Fanuc TP program (LS listing): ultrahose3.ls

/PROG  ultrahose3
/ATTR
COMMENT	= "19-03-19 19:07:18";
PROG_SIZE	= 0;
DEFAULT_GROUP	= 1, *, *, *, *;
/APPL
    ARC Welding Equipment: 1, *, *, *, *;
/MN
   1:  CALL HOME_ALL;
   1:  UFRAME_NUM = 1;
   1:  UTOOL_NUM = 3;
   1:  COL GUARD ADJUST 150;
   1:  PR[91] = PR[90];
   1:  PR[91,1] = PR[90,1] + -62.704;
   1:  PR[91,2] = PR[90,2] + 18.714;
   1:  PR[91,3] = PR[90,3] + 69.095;
   1:L PR[91] R[100]mm/sec CNT100;
   1:  PR[91,1] = PR[90,1] + -67.808;
   1:  PR[91,2] = PR[90,2] + 15.587;
   1:  PR[91,3] = PR[90,3] + 67.803;
   1:L PR[91] R[100]mm/sec CNT100;
   1:  PR[91,1] = PR[90,1] + -70.681;
   1:  PR[91,2] = PR[90,2] + 12.957;
   1:  PR[91,3] = PR[90,3] + 67.824;
   1:L PR[91] R[100]mm/sec CNT100;
   1:  PR[91,1] = PR[90,1] + -71.666;
   1:  PR[91,2] = PR[90,2] + 11.982;
   1:  PR[91,3] = PR[90,3] + 67.838;
   1:L PR[91] R[100]mm/sec CNT100;
   1:  PR[91,1] = PR[90,1] + -74.314;
   1:  PR[91,2] = PR[90,2] + 7.950;
   1:  PR[91,3] = PR[90,3] + 67.843;
   1:L PR[91] R[100]mm/sec CNT100;
   1:  PR[91,1] = PR[90,1] + -75.904;
   1:  PR[91,2] = PR[90,2] + 3.669;
   1:  PR[91,3] = PR[90,3] + 67.861;
   1:L PR[91] R[100]mm/sec CNT100;
   1:  PR[91,1] = PR[90,1] + -76.068;
   1:  PR[91,2] = PR[90,2] + 2.308;
   1:  PR[91,3] = PR[90,3] + 67.877;
   1:L PR[91] R[100]mm/sec CNT100;
   1:  PR[91,1] = PR[90,1] + -76.476;
   1:  PR[91,2] = PR[90,2] + 0.036;
   1:  PR[91,3] = PR[90,3] + 67.882;
   1:L PR[91] R[100]mm/sec CNT100;
   1:  PR[91,1] = PR[90,1] + -76.570;
   1:  PR[91,2] = PR[90,2] + -0.724;
   1:  PR[91,3] = PR[90,3] + 67.890;
   1:L PR[91] R[100]mm/sec CNT100;
   1:  PR[91,1] = PR[90,1] + -76.127;
   1:  PR[91,2] = PR[90,2] + -4.152;
   1:  PR[91,3] = PR[90,3] + 67.893;
   1:L PR[91] R[100]mm/sec CNT100;
   1:  PR[91,1] = PR[90,1] + -75.971;
   1:  PR[91,2] = PR[90,2] + -4.906;
   1:  PR[91,3] = PR[90,3] + 67.905;
   1:L PR[91] R[100]mm/sec CNT100;
   1:  PR[91,1] = PR[90,1] + -75.920;
   1:  PR[91,2] = PR[90,2] + -5.300;
   1:  PR[91,3] = PR[90,3] + 67.908;
   1:L PR[91] R[100]mm/sec CNT100;
   1:  PR[91,1] = PR[90,1] + -74.122;
   1:  PR[91,2] = PR[90,2] + -9.726;
   1:  PR[91,3] = PR[90,3] + 67.910;
   1:L PR[91] R[100]mm/sec CNT100;
   1:  PR[91,1] = PR[90,1] + -71.147;
   1:  PR[91,2] = PR[90,2] + -13.861;
   1:  PR[91,3] = PR[90,3] + 67.927;
   1:L PR[91] R[100]mm/sec CNT100;
   1:  PR[91,1] = PR[90,1] + -69.141;
   1:  PR[91,2] = PR[90,2] + -15.680;
   1:  PR[91,3] = PR[90,3] + 67.945;
   1:L PR[91] R[100]mm/sec CNT100;
   1:  PR[91,1] = PR[90,1] + -67.080;
   1:  PR[91,2] = PR[90,2] + -17.518;
   1:  PR[91,3] = PR[90,3] + 67.955;
   1:L PR[91] R[100]mm/sec CNT100;
   1:  PR[91,1] = PR[90,1] + -62.025;
   1:  PR[91,2] = PR[90,2] + -20.541;
   1:  PR[91,3] = PR[90,3] + 67.965;
   1:L PR[91] R[100]mm/sec CNT100;
   1:  PR[91,1] = PR[90,1] + -60.674;
   1:  PR[91,2] = PR[90,2] + -21.047;
   1:  PR[91,3] = PR[90,3] + 67.986;
   1:L PR[91] R[100]mm/sec CNT100;
   1:  PR[91,1] = PR[90,1] + -56.313;
   1:  PR[91,2] = PR[90,2] + -22.600;
   1:  PR[91,3] = PR[90,3] + 67.991;
   1:L PR[91] R[100]mm/sec CNT100;
   1:  PR[91,1] = PR[90,1] + -53.537;
   1:  PR[91,2] = PR[90,2] + -23.271;
   1:  PR[91,3] = PR[90,3] + 68.008;
   1:L PR[91] R[100]mm/sec CNT100;
   1:  PR[91,1] = PR[90,1] + -50.510;
   1:  PR[91,2] = PR[90,2] + -23.850;
   1:  PR[91,3] = PR[90,3] + 68.018;
   1:L PR[91] R[100]mm/sec CNT100;
   1:  PR[91,1] = PR[90,1] + -46.666;
   1:  PR[91,2] = PR[90,2] + -24.219;
   1:  PR[91,3] = PR[90,3] + 68.029;
   1:L PR[91] R[100]mm/sec CNT100;
   1:  PR[91,1] = PR[90,1] + -44.723;
   1:  PR[91,2] = PR[90,2] + -24.423;
   1:  PR[91,3] = PR[90,3] + 68.043;
   1:L PR[91] R[100]mm/sec CNT100;
   1:  PR[91,1] = PR[90,1] + -43.071;
   1:  PR[91,2] = PR[90,2] + -24.533;
   1:  PR[91,3] = PR[90,3] + 68.050;
   1:L PR[91] R[100]mm/sec CNT100;
   1:  PR[91,1] = PR[90,1] + -39.194;
   1:  PR[91,2] = PR[90,2] + -24.475;
   1:  PR[91,3] = PR[90,3] + 68.056;
   1:L PR[91] R[100]mm/sec CNT100;
   1:  PR[91,1] = PR[90,1] + -35.228;
   1:  PR[91,2] = PR[90,2] + -24.237;
   1:  PR[91,3] = PR[90,3] + 68.070;
   1:L PR[91] R[100]mm/sec CNT100;
   1:  PR[91,1] = PR[90,1] + -31.937;
   1:  PR[91,2] = PR[90,2] + -24.126;
   1:  PR[91,3] = PR[90,3] + 68.085;
   1:L PR[91] R[100]mm/sec CNT100;
   1:  PR[91,1] = PR[90,1] + -25.421;
   1:  PR[91,2] = PR[90,2] + -23.278;
   1:  PR[91,3] = PR[90,3] + 68.096;
   1:L PR[91] R[100]mm/sec CNT100;
   1:  PR[91,1] = PR[90,1] + -23.909;
   1:  PR[91,2] = PR[90,2] + -23.104;
   1:  PR[91,3] = PR[90,3] + 68.120;
   1:L PR[91] R[100]mm/sec CNT100;
   1:  PR[91,1] = PR[90,1] + -23.194;
   1:  PR[91,2] = PR[90,2] + -22.983;
   1:  PR[91,3] = PR[90,3] + 68.126;
   1:L PR[91] R[100]mm/sec CNT100;
   1:  PR[91,1] = PR[90,1] + -18.760;
   1:  PR[91,2] = PR[90,2] + -22.151;
   1:  PR[91,3] = PR[90,3] + 68.128;
   1:L PR[91] R[100]mm/sec CNT100;
   1:  PR[91,1] = PR[90,1] + -17.454;
   1:  PR[91,2] = PR[90,2] + -22.712;
   1:  PR[91,3] = PR[90,3] + 68.144;
   1:L PR[91] R[100]mm/sec CNT100;
   1:  PR[91,1] = PR[90,1] + -16.961;
   1:  PR[91,2] = PR[90,2] + -22.855;
   1:  PR[91,3] = PR[90,3] + 68.150;
   1:L PR[91] R[100]mm/sec CNT100;
   1:  PR[91,1] = PR[90,1] + -14.286;
   1:  PR[91,2] = PR[90,2] + -23.568;
   1:  PR[91,3] = PR[90,3] + 68.151;
   1:L PR[91] R[100]mm/sec CNT100;
   1:  PR[91,1] = PR[90,1] + -12.800;
   1:  PR[91,2] = PR[90,2] + -23.980;
   1:  PR[91,3] = PR[90,3] + 68.161;
   1:L PR[91] R[100]mm/sec CNT100;
   1:  PR[91,1] = PR[90,1] + -12.108;
   1:  PR[91,2] = PR[90,2] + -24.142;
   1:  PR[91,3] = PR[90,3] + 68.167;
   1:L PR[91] R[100]mm/sec CNT100;
   1:  PR[91,1] = PR[90,1] + -11.357;
   1:  PR[91,2] = PR[90,2] + -24.214;
   1:  PR[91,3] = PR[90,3] + 68.170;
   1:L PR[91] R[100]mm/sec CNT100;
   1:  PR[91,1] = PR[90,1] + -6.128;
   1:  PR[91,2] = PR[90,2] + -24.637;
   1:  PR[91,3] = PR[90,3] + 68.172;
   1:L PR[91] R[100]mm/sec CNT100;
   1:  PR[91,1] = PR[90,1] + -2.890;
   1:  PR[91,2] = PR[90,2] + -24.354;
   1:  PR[91,3] = PR[90,3] + 68.191;
   1:L PR[91] R[100]mm/sec CNT100;
   1:  PR[91,1] = PR[90,1] + -0.001;
   1:  PR[91,2] = PR[90,2] + -24.062;
   1:  PR[91,3] = PR[90,3] + 68.203;
   1:L PR[91] R[100]mm/sec CNT100;
   1:  PR[91,1] = PR[90,1] + 5.816;
   1:  PR[91,2] = PR[90,2] + -22.408;
   1:  PR[91,3] = PR[90,3] + 68.213;
   1:L PR[91] R[100]mm/sec CNT100;
   1:  PR[91,1] = PR[90,1] + 6.060;
   1:  PR[91,2] = PR[90,2] + -22.335;
   1:  PR[91,3] = PR[90,3] + 68.235;
   1:L PR[91] R[100]mm/sec CNT100;
   1:  PR[91,1] = PR[90,1] + 7.030;
   1:  PR[91,2] = PR[90,2] + -21.873;
   1:  PR[91,3] = PR[90,3] + 68.236;
   1:L PR[91] R[100]mm/sec CNT100;
   1:  PR[91,1] = PR[90,1] + 8.393;
   1:  PR[91,2] = PR[90,2] + -22.591;
   1:  PR[91,3] = PR[90,3] + 68.240;
   1:L PR[91] R[100]mm/sec CNT100;
   1:  PR[91,1] = PR[90,1] + 11.474;
   1:  PR[91,2] = PR[90,2] + -24.006;
   1:  PR[91,3] = PR[90,3] + 68.245;
   1:L PR[91] R[100]mm/sec CNT100;
   1:  PR[91,1] = PR[90,1] + 15.747;
   1:  PR[91,2] = PR[90,2] + -25.170;
   1:  PR[91,3] = PR[90,3] + 68.258;
   1:L PR[91] R[100]mm/sec CNT100;
   1:  PR[91,1] = PR[90,1] + 17.096;
   1:  PR[91,2] = PR[90,2] + -25.461;
   1:  PR[91,3] = PR[90,3] + 68.274;
   1:L PR[91] R[100]mm/sec CNT100;
   1:  PR[91,1] = PR[90,1] + 21.812;
   1:  PR[91,2] = PR[90,2] + -25.653;
   1:  PR[91,3] = PR[90,3] + 68.279;
   1:L PR[91] R[100]mm/sec CNT100;
   1:  PR[91,1] = PR[90,1] + 22.821;
   1:  PR[91,2] = PR[90,2] + -25.620;
   1:  PR[91,3] = PR[90,3] + 68.296;
   1:L PR[91] R[100]mm/sec CNT100;
   1:  PR[91,1] = PR[90,1] + 24.497;
   1:  PR[91,2] = PR[90,2] + -25.365;
   1:  PR[91,3] = PR[90,3] + 68.299;
   1:L PR[91] R[100]mm/sec CNT100;
   1:  PR[91,1] = PR[90,1] + 28.145;
   1:  PR[91,2] = PR[90,2] + -24.676;
   1:  PR[91,3] = PR[90,3] + 68.305;
   1:L PR[91] R[100]mm/sec CNT100;
   1:  PR[91,1] = PR[90,1] + 30.783;
   1:  PR[91,2] = PR[90,2] + -25.399;
   1:  PR[91,3] = PR[90,3] + 68.319;
   1:L PR[91] R[100]mm/sec CNT100;
   1:  PR[91,1] = PR[90,1] + 33.304;
   1:  PR[91,2] = PR[90,2] + -26.004;
   1:  PR[91,3] = PR[90,3] + 68.329;
   1:L PR[91] R[100]mm/sec CNT100;
   1:  PR[91,1] = PR[90,1] + 37.954;
   1:  PR[91,2] = PR[90,2] + -26.647;
   1:  PR[91,3] = PR[90,3] + 68.338;
   1:L PR[91] R[100]mm/sec CNT100;
   1:  PR[91,1] = PR[90,1] + 43.879;
   1:  PR[91,2] = PR[90,2] + -26.624;
   1:  PR[91,3] = PR[90,3] + 68.355;
   1:L PR[91] R[100]mm/sec CNT100;
   1:  PR[91,1] = PR[90,1] + 49.043;
   1:  PR[91,2] = PR[90,2] + -26.009;
   1:  PR[91,3] = PR[90,3] + 68.376;
   1:L PR[91] R[100]mm/sec CNT100;
   1:  PR[91,1] = PR[90,1] + 53.583;
   1:  PR[91,2] = PR[90,2] + -25.090;
   1:  PR[91,3] = PR[90,3] + 68.395;
   1:L PR[91] R[100]mm/sec CNT100;
   1:  PR[91,1] = PR[90,1] + 55.197;
   1:  PR[91,2] = PR[90,2] + -24.588;
   1:  PR[91,3] = PR[90,3] + 68.411;
   1:L PR[91] R[100]mm/sec CNT100;
   1:  PR[91,1] = PR[90,1] + 59.058;
   1:  PR[91,2] = PR[90,2] + -23.334;
   1:  PR[91,3] = PR[90,3] + 68.418;
   1:L PR[91] R[100]mm/sec CNT100;
   1:  PR[91,1] = PR[90,1] + 61.784;
   1:  PR[91,2] = PR[90,2] + -22.074;
   1:  PR[91,3] = PR[90,3] + 68.432;
   1:L PR[91] R[100]mm/sec CNT100;
   1:  PR[91,1] = PR[90,1] + 65.680;
   1:  PR[91,2] = PR[90,2] + -19.965;
   1:  PR[91,3] = PR[90,3] + 68.443;
   1:L PR[91] R[100]mm/sec CNT100;
   1:  PR[91,1] = PR[90,1] + 66.517;
   1:  PR[91,2] = PR[90,2] + -19.431;
   1:  PR[91,3] = PR[90,3] + 68.459;
   1:L PR[91] R[100]mm/sec CNT100;
   1:  PR[91,1] = PR[90,1] + 69.227;
   1:  PR[91,2] = PR[90,2] + -17.197;
   1:  PR[91,3] = PR[90,3] + 68.463;
   1:L PR[91] R[100]mm/sec CNT100;
   1:  PR[91,1] = PR[90,1] + 71.107;
   1:  PR[91,2] = PR[90,2] + -15.516;
   1:  PR[91,3] = PR[90,3] + 68.475;
   1:L PR[91] R[100]mm/sec CNT100;
   1:  PR[91,1] = PR[90,1] + 74.460;
   1:  PR[91,2] = PR[90,2] + -10.836;
   1:  PR[91,3] = PR[90,3] + 68.484;
   1:L PR[91] R[100]mm/sec CNT100;
   1:  PR[91,1] = PR[90,1] + 76.466;
   1:  PR[91,2] = PR[90,2] + -5.850;
   1:  PR[91,3] = PR[90,3] + 68.505;
   1:L PR[91] R[100]mm/sec CNT100;
   1:  PR[91,1] = PR[90,1] + 76.772;
   1:  PR[91,2] = PR[90,2] + -3.531;
   1:  PR[91,3] = PR[90,3] + 68.524;
   1:L PR[91] R[100]mm/sec CNT100;
   1:  PR[91,1] = PR[90,1] + 77.227;
   1:  PR[91,2] = PR[90,2] + -0.700;
   1:  PR[91,3] = PR[90,3] + 68.533;
   1:L PR[91] R[100]mm/sec CNT100;
   1:  PR[91,1] = PR[90,1] + 77.051;
   1:  PR[91,2] = PR[90,2] + 0.647;
   1:  PR[91,3] = PR[90,3] + 68.543;
   1:L PR[91] R[100]mm/sec CNT100;
   1:  PR[91,1] = PR[90,1] + 76.850;
   1:  PR[91,2] = PR[90,2] + 1.446;
   1:  PR[91,3] = PR[90,3] + 68.548;
   1:L PR[91] R[100]mm/sec CNT100;
   1:  PR[91,1] = PR[90,1] + 76.465;
   1:  PR[91,2] = PR[90,2] + 4.394;
   1:  PR[91,3] = PR[90,3] + 68.551;
   1:L PR[91] R[100]mm/sec CNT100;
   1:  PR[91,1] = PR[90,1] + 74.460;
   1:  PR[91,2] = PR[90,2] + 9.378;
   1:  PR[91,3] = PR[90,3] + 68.562;
   1:L PR[91] R[100]mm/sec CNT100;
   1:  PR[91,1] = PR[90,1] + 71.112;
   1:  PR[91,2] = PR[90,2] + 14.052;
   1:  PR[91,3] = PR[90,3] + 68.581;
   1:L PR[91] R[100]mm/sec CNT100;
   1:  PR[91,1] = PR[90,1] + 69.227;
   1:  PR[91,2] = PR[90,2] + 15.739;
   1:  PR[91,3] = PR[90,3] + 68.602;
   1:L PR[91] R[100]mm/sec CNT100;
   1:  PR[91,1] = PR[90,1] + 66.528;
   1:  PR[91,2] = PR[90,2] + 17.965;
   1:  PR[91,3] = PR[90,3] + 68.611;
   1:L PR[91] R[100]mm/sec CNT100;
   1:  PR[91,1] = PR[90,1] + 65.694;
   1:  PR[91,2] = PR[90,2] + 18.497;
   1:  PR[91,3] = PR[90,3] + 68.623;
   1:L PR[91] R[100]mm/sec CNT100;
   1:  PR[91,1] = PR[90,1] + 61.792;
   1:  PR[91,2] = PR[90,2] + 20.612;
   1:  PR[91,3] = PR[90,3] + 68.627;
   1:L PR[91] R[100]mm/sec CNT100;
   1:  PR[91,1] = PR[90,1] + 59.065;
   1:  PR[91,2] = PR[90,2] + 21.873;
   1:  PR[91,3] = PR[90,3] + 68.643;
   1:L PR[91] R[100]mm/sec CNT100;
   1:  PR[91,1] = PR[90,1] + 55.197;
   1:  PR[91,2] = PR[90,2] + 23.129;
   1:  PR[91,3] = PR[90,3] + 68.654;
   1:L PR[91] R[100]mm/sec CNT100;
   1:  PR[91,1] = PR[90,1] + 53.583;
   1:  PR[91,2] = PR[90,2] + 23.631;
   1:  PR[91,3] = PR[90,3] + 68.668;
   1:L PR[91] R[100]mm/sec CNT100;
   1:  PR[91,1] = PR[90,1] + 49.043;
   1:  PR[91,2] = PR[90,2] + 24.550;
   1:  PR[91,3] = PR[90,3] + 68.675;
   1:L PR[91] R[100]mm/sec CNT100;
   1:  PR[91,1] = PR[90,1] + 43.879;
   1:  PR[91,2] = PR[90,2] + 25.165;
   1:  PR[91,3] = PR[90,3] + 68.691;
   1:L PR[91] R[100]mm/sec CNT100;
   1:  PR[91,1] = PR[90,1] + 37.958;
   1:  PR[91,2] = PR[90,2] + 25.189;
   1:  PR[91,3] = PR[90,3] + 68.710;
   1:L PR[91] R[100]mm/sec CNT100;
   1:  PR[91,1] = PR[90,1] + 33.304;
   1:  PR[91,2] = PR[90,2] + 24.545;
   1:  PR[91,3] = PR[90,3] + 68.731;
   1:L PR[91] R[100]mm/sec CNT100;
   1:  PR[91,1] = PR[90,1] + 30.783;
   1:  PR[91,2] = PR[90,2] + 23.940;
   1:  PR[91,3] = PR[90,3] + 68.748;
   1:L PR[91] R[100]mm/sec CNT100;
   1:  PR[91,1] = PR[90,1] + 28.145;
   1:  PR[91,2] = PR[90,2] + 23.217;
   1:  PR[91,3] = PR[90,3] + 68.758;
   1:L PR[91] R[100]mm/sec CNT100;
   1:  PR[91,1] = PR[90,1] + 24.496;
   1:  PR[91,2] = PR[90,2] + 23.906;
   1:  PR[91,3] = PR[90,3] + 68.767;
   1:L PR[91] R[100]mm/sec CNT100;
   1:  PR[91,1] = PR[90,1] + 22.831;
   1:  PR[91,2] = PR[90,2] + 24.160;
   1:  PR[91,3] = PR[90,3] + 68.781;
   1:L PR[91] R[100]mm/sec CNT100;
   1:  PR[91,1] = PR[90,1] + 21.811;
   1:  PR[91,2] = PR[90,2] + 24.194;
   1:  PR[91,3] = PR[90,3] + 68.787;
   1:L PR[91] R[100]mm/sec CNT100;
   1:  PR[91,1] = PR[90,1] + 17.094;
   1:  PR[91,2] = PR[90,2] + 24.002;
   1:  PR[91,3] = PR[90,3] + 68.791;
   1:L PR[91] R[100]mm/sec CNT100;
   1:  PR[91,1] = PR[90,1] + 15.746;
   1:  PR[91,2] = PR[90,2] + 23.711;
   1:  PR[91,3] = PR[90,3] + 68.808;
   1:L PR[91] R[100]mm/sec CNT100;
   1:  PR[91,1] = PR[90,1] + 11.472;
   1:  PR[91,2] = PR[90,2] + 22.546;
   1:  PR[91,3] = PR[90,3] + 68.812;
   1:L PR[91] R[100]mm/sec CNT100;
   1:  PR[91,1] = PR[90,1] + 8.412;
   1:  PR[91,2] = PR[90,2] + 21.143;
   1:  PR[91,3] = PR[90,3] + 68.828;
   1:L PR[91] R[100]mm/sec CNT100;
   1:  PR[91,1] = PR[90,1] + 7.033;
   1:  PR[91,2] = PR[90,2] + 20.424;
   1:  PR[91,3] = PR[90,3] + 68.841;
   1:L PR[91] R[100]mm/sec CNT100;
   1:  PR[91,1] = PR[90,1] + 6.058;
   1:  PR[91,2] = PR[90,2] + 20.878;
   1:  PR[91,3] = PR[90,3] + 68.846;
   1:L PR[91] R[100]mm/sec CNT100;
   1:  PR[91,1] = PR[90,1] + 5.788;
   1:  PR[91,2] = PR[90,2] + 20.959;
   1:  PR[91,3] = PR[90,3] + 68.850;
   1:L PR[91] R[100]mm/sec CNT100;
   1:  PR[91,1] = PR[90,1] + 0.034;
   1:  PR[91,2] = PR[90,2] + 22.597;
   1:  PR[91,3] = PR[90,3] + 68.851;
   1:L PR[91] R[100]mm/sec CNT100;
   1:  PR[91,1] = PR[90,1] + -2.850;
   1:  PR[91,2] = PR[90,2] + 22.890;
   1:  PR[91,3] = PR[90,3] + 68.873;
   1:L PR[91] R[100]mm/sec CNT100;
   1:  PR[91,1] = PR[90,1] + -6.112;
   1:  PR[91,2] = PR[90,2] + 23.178;
   1:  PR[91,3] = PR[90,3] + 68.883;
   1:L PR[91] R[100]mm/sec CNT100;
   1:  PR[91,1] = PR[90,1] + -11.344;
   1:  PR[91,2] = PR[90,2] + 22.757;
   1:  PR[91,3] = PR[90,3] + 68.895;
   1:L PR[91] R[100]mm/sec CNT100;
   1:  PR[91,1] = PR[90,1] + -12.102;
   1:  PR[91,2] = PR[90,2] + 22.684;
   1:  PR[91,3] = PR[90,3] + 68.914;
   1:L PR[91] R[100]mm/sec CNT100;
   1:  PR[91,1] = PR[90,1] + -12.809;
   1:  PR[91,2] = PR[90,2] + 22.518;
   1:  PR[91,3] = PR[90,3] + 68.916;
   1:L PR[91] R[100]mm/sec CNT100;
   1:  PR[91,1] = PR[90,1] + -14.290;
   1:  PR[91,2] = PR[90,2] + 22.107;
   1:  PR[91,3] = PR[90,3] + 68.919;
   1:L PR[91] R[100]mm/sec CNT100;
   1:  PR[91,1] = PR[90,1] + -16.962;
   1:  PR[91,2] = PR[90,2] + 21.395;
   1:  PR[91,3] = PR[90,3] + 68.925;
   1:L PR[91] R[100]mm/sec CNT100;
   1:  PR[91,1] = PR[90,1] + -17.452;
   1:  PR[91,2] = PR[90,2] + 21.253;
   1:  PR[91,3] = PR[90,3] + 68.935;
   1:L PR[91] R[100]mm/sec CNT100;
   1:  PR[91,1] = PR[90,1] + -18.760;
   1:  PR[91,2] = PR[90,2] + 20.692;
   1:  PR[91,3] = PR[90,3] + 68.936;
   1:L PR[91] R[100]mm/sec CNT100;
   1:  PR[91,1] = PR[90,1] + -23.191;
   1:  PR[91,2] = PR[90,2] + 21.523;
   1:  PR[91,3] = PR[90,3] + 68.942;
   1:L PR[91] R[100]mm/sec CNT100;
   1:  PR[91,1] = PR[90,1] + -23.903;
   1:  PR[91,2] = PR[90,2] + 21.644;
   1:  PR[91,3] = PR[90,3] + 68.958;
   1:L PR[91] R[100]mm/sec CNT100;
   1:  PR[91,1] = PR[90,1] + -25.418;
   1:  PR[91,2] = PR[90,2] + 21.819;
   1:  PR[91,3] = PR[90,3] + 68.960;
   1:L PR[91] R[100]mm/sec CNT100;
   1:  PR[91,1] = PR[90,1] + -32.341;
   1:  PR[91,2] = PR[90,2] + 22.697;
   1:  PR[91,3] = PR[90,3] + 68.966;
   1:L PR[91] R[100]mm/sec CNT100;
   1:  PR[91,1] = PR[90,1] + -34.160;
   1:  PR[91,2] = PR[90,2] + 22.753;
   1:  PR[91,3] = PR[90,3] + 68.991;
   1:L PR[91] R[100]mm/sec CNT100;
   1:  PR[91,1] = PR[90,1] + -39.829;
   1:  PR[91,2] = PR[90,2] + 23.076;
   1:  PR[91,3] = PR[90,3] + 68.998;
   1:L PR[91] R[100]mm/sec CNT100;
   1:  PR[91,1] = PR[90,1] + -44.279;
   1:  PR[91,2] = PR[90,2] + 22.883;
   1:  PR[91,3] = PR[90,3] + 69.018;
   1:L PR[91] R[100]mm/sec CNT100;
   1:  PR[91,1] = PR[90,1] + -46.346;
   1:  PR[91,2] = PR[90,2] + 22.848;
   1:  PR[91,3] = PR[90,3] + 69.034;
   1:L PR[91] R[100]mm/sec CNT100;
   1:  PR[91,1] = PR[90,1] + -47.984;
   1:  PR[91,2] = PR[90,2] + 22.746;
   1:  PR[91,3] = PR[90,3] + 69.042;
   1:L PR[91] R[100]mm/sec CNT100;
   1:  PR[91,1] = PR[90,1] + -51.432;
   1:  PR[91,2] = PR[90,2] + 22.175;
   1:  PR[91,3] = PR[90,3] + 69.047;
   1:L PR[91] R[100]mm/sec CNT100;
   1:  PR[91,1] = PR[90,1] + -56.575;
   1:  PR[91,2] = PR[90,2] + 21.118;
   1:  PR[91,3] = PR[90,3] + 69.060;
   1:L PR[91] R[100]mm/sec CNT100;
   1:  PR[91,1] = PR[90,1] + -56.591;
   1:  PR[91,2] = PR[90,2] + 21.114;
   1:  PR[91,3] = PR[90,3] + 69.079;
   1:L PR[91] R[100]mm/sec CNT100;
   1:  PR[91,1] = PR[90,1] + -60.733;
   1:  PR[91,2] = PR[90,2] + 19.500;
   1:L PR[91] R[100]mm/sec CNT100;
   1:  PR[91] = PR[90];
   1:  PR[91,1] = PR[90,1] + -66.757;
   1:  PR[91,2] = PR[90,2] + 15.737;
   1:  PR[91,3] = PR[90,3] + 70.395;
   1:L PR[91] R[100]mm/sec CNT100;
   1:  PR[91,1] = PR[90,1] + -70.803;
   1:  PR[91,2] = PR[90,2] + 12.036;
   1:  PR[91,3] = PR[90,3] + 69.117;
   1:L PR[91] R[100]mm/sec CNT100;
   1:  PR[91,1] = PR[90,1] + -72.056;
   1:  PR[91,2] = PR[90,2] + 10.273;
   1:  PR[91,3] = PR[90,3] + 69.137;
   1:L PR[91] R[100]mm/sec CNT100;
   1:  PR[91,1] = PR[90,1] + -73.534;
   1:  PR[91,2] = PR[90,2] + 8.022;
   1:  PR[91,3] = PR[90,3] + 69.145;
   1:L PR[91] R[100]mm/sec CNT100;
   1:  PR[91,1] = PR[90,1] + -75.139;
   1:  PR[91,2] = PR[90,2] + 3.706;
   1:  PR[91,3] = PR[90,3] + 69.155;
   1:L PR[91] R[100]mm/sec CNT100;
   1:  PR[91,1] = PR[90,1] + -75.226;
   1:  PR[91,2] = PR[90,2] + 2.985;
   1:  PR[91,3] = PR[90,3] + 69.171;
   1:L PR[91] R[100]mm/sec CNT100;
   1:  PR[91,1] = PR[90,1] + -75.465;
   1:  PR[91,2] = PR[90,2] + 1.656;
   1:  PR[91,3] = PR[90,3] + 69.174;
   1:L PR[91] R[100]mm/sec CNT100;
   1:  PR[91,1] = PR[90,1] + -75.759;
   1:  PR[91,2] = PR[90,2] + -0.724;
   1:  PR[91,3] = PR[90,3] + 69.179;
   1:L PR[91] R[100]mm/sec CNT100;
   1:  PR[91,1] = PR[90,1] + -75.499;
   1:  PR[91,2] = PR[90,2] + -2.738;
   1:  PR[91,3] = PR[90,3] + 69.188;
   1:L PR[91] R[100]mm/sec CNT100;
   1:  PR[91,1] = PR[90,1] + -75.172;
   1:  PR[91,2] = PR[90,2] + -4.310;
   1:  PR[91,3] = PR[90,3] + 69.195;
   1:L PR[91] R[100]mm/sec CNT100;
   1:  PR[91,1] = PR[90,1] + -75.041;
   1:  PR[91,2] = PR[90,2] + -5.328;
   1:  PR[91,3] = PR[90,3] + 69.201;
   1:L PR[91] R[100]mm/sec CNT100;
   1:  PR[91,1] = PR[90,1] + -73.235;
   1:  PR[91,2] = PR[90,2] + -9.782;
   1:  PR[91,3] = PR[90,3] + 69.205;
   1:L PR[91] R[100]mm/sec CNT100;
   1:  PR[91,1] = PR[90,1] + -70.249;
   1:  PR[91,2] = PR[90,2] + -13.943;
   1:  PR[91,3] = PR[90,3] + 69.222;
   1:L PR[91] R[100]mm/sec CNT100;
   1:  PR[91,1] = PR[90,1] + -67.479;
   1:  PR[91,2] = PR[90,2] + -16.454;
   1:  PR[91,3] = PR[90,3] + 69.241;
   1:L PR[91] R[100]mm/sec CNT100;
   1:  PR[91,1] = PR[90,1] + -66.164;
   1:  PR[91,2] = PR[90,2] + -17.628;
   1:  PR[91,3] = PR[90,3] + 69.254;
   1:L PR[91] R[100]mm/sec CNT100;
   1:  PR[91,1] = PR[90,1] + -61.781;
   1:  PR[91,2] = PR[90,2] + -20.254;
   1:  PR[91,3] = PR[90,3] + 69.261;
   1:L PR[91] R[100]mm/sec CNT100;
   1:  PR[91,1] = PR[90,1] + -61.089;
   1:  PR[91,2] = PR[90,2] + -20.640;
   1:  PR[91,3] = PR[90,3] + 69.279;
   1:L PR[91] R[100]mm/sec CNT100;
   1:  PR[91,1] = PR[90,1] + -60.787;
   1:  PR[91,2] = PR[90,2] + -20.763;
   1:  PR[91,3] = PR[90,3] + 69.282;
   1:L PR[91] R[100]mm/sec CNT100;
   1:  PR[91,1] = PR[90,1] + -55.434;
   1:  PR[91,2] = PR[90,2] + -22.669;
   1:  PR[91,3] = PR[90,3] + 69.283;
   1:L PR[91] R[100]mm/sec CNT100;
   1:  PR[91,1] = PR[90,1] + -51.154;
   1:  PR[91,2] = PR[90,2] + -23.704;
   1:  PR[91,3] = PR[90,3] + 69.304;
   1:L PR[91] R[100]mm/sec CNT100;
   1:  PR[91,1] = PR[90,1] + -49.687;
   1:  PR[91,2] = PR[90,2] + -23.984;
   1:  PR[91,3] = PR[90,3] + 69.320;
   1:L PR[91] R[100]mm/sec CNT100;
   1:  PR[91,1] = PR[90,1] + -47.779;
   1:  PR[91,2] = PR[90,2] + -24.167;
   1:  PR[91,3] = PR[90,3] + 69.326;
   1:L PR[91] R[100]mm/sec CNT100;
   1:  PR[91,1] = PR[90,1] + -43.981;
   1:  PR[91,2] = PR[90,2] + -24.566;
   1:  PR[91,3] = PR[90,3] + 69.333;
   1:L PR[91] R[100]mm/sec CNT100;
   1:  PR[91,1] = PR[90,1] + -40.665;
   1:  PR[91,2] = PR[90,2] + -24.787;
   1:  PR[91,3] = PR[90,3] + 69.346;
   1:L PR[91] R[100]mm/sec CNT100;
   1:  PR[91,1] = PR[90,1] + -38.425;
   1:  PR[91,2] = PR[90,2] + -24.754;
   1:  PR[91,3] = PR[90,3] + 69.358;
   1:L PR[91] R[100]mm/sec CNT100;
   1:  PR[91,1] = PR[90,1] + -36.087;
   1:  PR[91,2] = PR[90,2] + -24.613;
   1:  PR[91,3] = PR[90,3] + 69.367;
   1:L PR[91] R[100]mm/sec CNT100;
   1:  PR[91,1] = PR[90,1] + -32.395;
   1:  PR[91,2] = PR[90,2] + -24.500;
   1:  PR[91,3] = PR[90,3] + 69.375;
   1:L PR[91] R[100]mm/sec CNT100;
   1:  PR[91,1] = PR[90,1] + -29.764;
   1:  PR[91,2] = PR[90,2] + -24.400;
   1:  PR[91,3] = PR[90,3] + 69.389;
   1:L PR[91] R[100]mm/sec CNT100;
   1:  PR[91,1] = PR[90,1] + -26.068;
   1:  PR[91,2] = PR[90,2] + -23.919;
   1:  PR[91,3] = PR[90,3] + 69.398;
   1:L PR[91] R[100]mm/sec CNT100;
   1:  PR[91,1] = PR[90,1] + -22.104;
   1:  PR[91,2] = PR[90,2] + -23.469;
   1:  PR[91,3] = PR[90,3] + 69.412;
   1:L PR[91] R[100]mm/sec CNT100;
   1:  PR[91,1] = PR[90,1] + -21.916;
   1:  PR[91,2] = PR[90,2] + -23.463;
   1:  PR[91,3] = PR[90,3] + 69.426;
   1:L PR[91] R[100]mm/sec CNT100;
   1:  PR[91,1] = PR[90,1] + -20.919;
   1:  PR[91,2] = PR[90,2] + -23.327;
   1:  PR[91,3] = PR[90,3] + 69.427;
   1:L PR[91] R[100]mm/sec CNT100;
   1:  PR[91,1] = PR[90,1] + -17.354;
   1:  PR[91,2] = PR[90,2] + -22.716;
   1:  PR[91,3] = PR[90,3] + 69.431;
   1:L PR[91] R[100]mm/sec CNT100;
   1:  PR[91,1] = PR[90,1] + -16.762;
   1:  PR[91,2] = PR[90,2] + -22.935;
   1:  PR[91,3] = PR[90,3] + 69.444;
   1:L PR[91] R[100]mm/sec CNT100;
   1:  PR[91,1] = PR[90,1] + -13.178;
   1:  PR[91,2] = PR[90,2] + -23.926;
   1:  PR[91,3] = PR[90,3] + 69.446;
   1:L PR[91] R[100]mm/sec CNT100;
   1:  PR[91,1] = PR[90,1] + -11.411;
   1:  PR[91,2] = PR[90,2] + -24.340;
   1:  PR[91,3] = PR[90,3] + 69.460;
   1:L PR[91] R[100]mm/sec CNT100;
   1:  PR[91,1] = PR[90,1] + -9.538;
   1:  PR[91,2] = PR[90,2] + -24.521;
   1:  PR[91,3] = PR[90,3] + 69.466;
   1:L PR[91] R[100]mm/sec CNT100;
   1:  PR[91,1] = PR[90,1] + -5.371;
   1:  PR[91,2] = PR[90,2] + -24.857;
   1:  PR[91,3] = PR[90,3] + 69.473;
   1:L PR[91] R[100]mm/sec CNT100;
   1:  PR[91,1] = PR[90,1] + -0.893;
   1:  PR[91,2] = PR[90,2] + -24.466;
   1:  PR[91,3] = PR[90,3] + 69.488;
   1:L PR[91] R[100]mm/sec CNT100;
   1:  PR[91,1] = PR[90,1] + 0.829;
   1:  PR[91,2] = PR[90,2] + -24.292;
   1:  PR[91,3] = PR[90,3] + 69.505;
   1:L PR[91] R[100]mm/sec CNT100;
   1:  PR[91,1] = PR[90,1] + 5.257;
   1:  PR[91,2] = PR[90,2] + -23.033;
   1:  PR[91,3] = PR[90,3] + 69.511;
   1:L PR[91] R[100]mm/sec CNT100;
   1:  PR[91,1] = PR[90,1] + 7.503;
   1:  PR[91,2] = PR[90,2] + -22.456;
   1:  PR[91,3] = PR[90,3] + 69.528;
   1:L PR[91] R[100]mm/sec CNT100;
   1:  PR[91,1] = PR[90,1] + 11.340;
   1:  PR[91,2] = PR[90,2] + -24.218;
   1:  PR[91,3] = PR[90,3] + 69.536;
   1:L PR[91] R[100]mm/sec CNT100;
   1:  PR[91,1] = PR[90,1] + 15.050;
   1:  PR[91,2] = PR[90,2] + -25.228;
   1:  PR[91,3] = PR[90,3] + 69.551;
   1:L PR[91] R[100]mm/sec CNT100;
   1:  PR[91,1] = PR[90,1] + 17.058;
   1:  PR[91,2] = PR[90,2] + -25.662;
   1:  PR[91,3] = PR[90,3] + 69.565;
   1:L PR[91] R[100]mm/sec CNT100;
   1:  PR[91,1] = PR[90,1] + 21.206;
   1:  PR[91,2] = PR[90,2] + -25.830;
   1:  PR[91,3] = PR[90,3] + 69.573;
   1:L PR[91] R[100]mm/sec CNT100;
   1:  PR[91,1] = PR[90,1] + 22.871;
   1:  PR[91,2] = PR[90,2] + -25.776;
   1:  PR[91,3] = PR[90,3] + 69.588;
   1:L PR[91] R[100]mm/sec CNT100;
   1:  PR[91,1] = PR[90,1] + 25.545;
   1:  PR[91,2] = PR[90,2] + -25.370;
   1:  PR[91,3] = PR[90,3] + 69.594;
   1:L PR[91] R[100]mm/sec CNT100;
   1:  PR[91,1] = PR[90,1] + 27.613;
   1:  PR[91,2] = PR[90,2] + -24.979;
   1:  PR[91,3] = PR[90,3] + 69.604;
   1:L PR[91] R[100]mm/sec CNT100;
   1:  PR[91,1] = PR[90,1] + 29.163;
   1:  PR[91,2] = PR[90,2] + -25.404;
   1:  PR[91,3] = PR[90,3] + 69.612;
   1:L PR[91] R[100]mm/sec CNT100;
   1:  PR[91,1] = PR[90,1] + 32.825;
   1:  PR[91,2] = PR[90,2] + -26.283;
   1:  PR[91,3] = PR[90,3] + 69.617;
   1:L PR[91] R[100]mm/sec CNT100;
   1:  PR[91,1] = PR[90,1] + 36.431;
   1:  PR[91,2] = PR[90,2] + -26.781;
   1:  PR[91,3] = PR[90,3] + 69.631;
   1:L PR[91] R[100]mm/sec CNT100;
   1:  PR[91,1] = PR[90,1] + 37.530;
   1:  PR[91,2] = PR[90,2] + -26.871;
   1:  PR[91,3] = PR[90,3] + 69.644;
   1:L PR[91] R[100]mm/sec CNT100;
   1:  PR[91,1] = PR[90,1] + 39.448;
   1:  PR[91,2] = PR[90,2] + -26.838;
   1:  PR[91,3] = PR[90,3] + 69.648;
   1:L PR[91] R[100]mm/sec CNT100;
   1:  PR[91,1] = PR[90,1] + 42.921;
   1:  PR[91,2] = PR[90,2] + -26.825;
   1:  PR[91,3] = PR[90,3] + 69.655;
   1:L PR[91] R[100]mm/sec CNT100;
   1:  PR[91,1] = PR[90,1] + 46.083;
   1:  PR[91,2] = PR[90,2] + -26.444;
   1:  PR[91,3] = PR[90,3] + 69.668;
   1:L PR[91] R[100]mm/sec CNT100;
   1:  PR[91,1] = PR[90,1] + 48.210;
   1:  PR[91,2] = PR[90,2] + -26.159;
   1:  PR[91,3] = PR[90,3] + 69.680;
   1:L PR[91] R[100]mm/sec CNT100;
   1:  PR[91,1] = PR[90,1] + 49.893;
   1:  PR[91,2] = PR[90,2] + -25.741;
   1:  PR[91,3] = PR[90,3] + 69.687;
   1:L PR[91] R[100]mm/sec CNT100;
   1:  PR[91,1] = PR[90,1] + 52.863;
   1:  PR[91,2] = PR[90,2] + -25.134;
   1:  PR[91,3] = PR[90,3] + 69.694;
   1:L PR[91] R[100]mm/sec CNT100;
   1:  PR[91,1] = PR[90,1] + 56.392;
   1:  PR[91,2] = PR[90,2] + -24.037;
   1:  PR[91,3] = PR[90,3] + 69.705;
   1:L PR[91] R[100]mm/sec CNT100;
   1:  PR[91,1] = PR[90,1] + 57.694;
   1:  PR[91,2] = PR[90,2] + -23.615;
   1:  PR[91,3] = PR[90,3] + 69.718;
   1:L PR[91] R[100]mm/sec CNT100;
   1:  PR[91,1] = PR[90,1] + 61.193;
   1:  PR[91,2] = PR[90,2] + -21.997;
   1:  PR[91,3] = PR[90,3] + 69.723;
   1:L PR[91] R[100]mm/sec CNT100;
   1:  PR[91,1] = PR[90,1] + 64.047;
   1:  PR[91,2] = PR[90,2] + -20.453;
   1:  PR[91,3] = PR[90,3] + 69.737;
   1:L PR[91] R[100]mm/sec CNT100;
   1:  PR[91,1] = PR[90,1] + 65.701;
   1:  PR[91,2] = PR[90,2] + -19.397;
   1:  PR[91,3] = PR[90,3] + 69.749;
   1:L PR[91] R[100]mm/sec CNT100;
   1:  PR[91,1] = PR[90,1] + 70.308;
   1:  PR[91,2] = PR[90,2] + -15.595;
   1:  PR[91,3] = PR[90,3] + 69.756;
   1:L PR[91] R[100]mm/sec CNT100;
   1:  PR[91,1] = PR[90,1] + 70.437;
   1:  PR[91,2] = PR[90,2] + -15.431;
   1:  PR[91,3] = PR[90,3] + 69.778;
   1:L PR[91] R[100]mm/sec CNT100;
   1:  PR[91,1] = PR[90,1] + 73.660;
   1:  PR[91,2] = PR[90,2] + -10.936;
   1:  PR[91,3] = PR[90,3] + 69.779;
   1:L PR[91] R[100]mm/sec CNT100;
   1:  PR[91,1] = PR[90,1] + 75.688;
   1:  PR[91,2] = PR[90,2] + -5.901;
   1:  PR[91,3] = PR[90,3] + 69.799;
   1:L PR[91] R[100]mm/sec CNT100;
   1:  PR[91,1] = PR[90,1] + 75.896;
   1:  PR[91,2] = PR[90,2] + -4.318;
   1:  PR[91,3] = PR[90,3] + 69.819;
   1:L PR[91] R[100]mm/sec CNT100;
   1:  PR[91,1] = PR[90,1] + 76.478;
   1:  PR[91,2] = PR[90,2] + -0.700;
   1:  PR[91,3] = PR[90,3] + 69.824;
   1:L PR[91] R[100]mm/sec CNT100;
   1:  PR[91,1] = PR[90,1] + 76.413;
   1:  PR[91,2] = PR[90,2] + -0.209;
   1:  PR[91,3] = PR[90,3] + 69.838;
   1:L PR[91] R[100]mm/sec CNT100;
   1:  PR[91,1] = PR[90,1] + 76.165;
   1:  PR[91,2] = PR[90,2] + 0.777;
   1:  PR[91,3] = PR[90,3] + 69.839;
   1:L PR[91] R[100]mm/sec CNT100;
   1:  PR[91,1] = PR[90,1] + 75.687;
   1:  PR[91,2] = PR[90,2] + 4.444;
   1:  PR[91,3] = PR[90,3] + 69.843;
   1:L PR[91] R[100]mm/sec CNT100;
   1:  PR[91,1] = PR[90,1] + 73.661;
   1:  PR[91,2] = PR[90,2] + 9.475;
   1:  PR[91,3] = PR[90,3] + 69.857;
   1:L PR[91] R[100]mm/sec CNT100;
   1:  PR[91,1] = PR[90,1] + 70.437;
   1:  PR[91,2] = PR[90,2] + 13.974;
   1:  PR[91,3] = PR[90,3] + 69.876;
   1:L PR[91] R[100]mm/sec CNT100;
   1:  PR[91,1] = PR[90,1] + 70.316;
   1:  PR[91,2] = PR[90,2] + 14.128;
   1:  PR[91,3] = PR[90,3] + 69.896;
   1:L PR[91] R[100]mm/sec CNT100;
   1:  PR[91,1] = PR[90,1] + 65.710;
   1:  PR[91,2] = PR[90,2] + 17.932;
   1:  PR[91,3] = PR[90,3] + 69.897;
   1:L PR[91] R[100]mm/sec CNT100;
   1:  PR[91,1] = PR[90,1] + 64.057;
   1:  PR[91,2] = PR[90,2] + 18.987;
   1:  PR[91,3] = PR[90,3] + 69.919;
   1:L PR[91] R[100]mm/sec CNT100;
   1:  PR[91,1] = PR[90,1] + 61.200;
   1:  PR[91,2] = PR[90,2] + 20.536;
   1:  PR[91,3] = PR[90,3] + 69.926;
   1:L PR[91] R[100]mm/sec CNT100;
   1:  PR[91,1] = PR[90,1] + 57.697;
   1:  PR[91,2] = PR[90,2] + 22.155;
   1:  PR[91,3] = PR[90,3] + 69.938;
   1:L PR[91] R[100]mm/sec CNT100;
   1:  PR[91,1] = PR[90,1] + 56.393;
   1:  PR[91,2] = PR[90,2] + 22.578;
   1:  PR[91,3] = PR[90,3] + 69.952;
   1:L PR[91] R[100]mm/sec CNT100;
   1:  PR[91,1] = PR[90,1] + 52.863;
   1:  PR[91,2] = PR[90,2] + 23.675;
   1:  PR[91,3] = PR[90,3] + 69.957;
   1:L PR[91] R[100]mm/sec CNT100;
   1:  PR[91,1] = PR[90,1] + 49.893;
   1:  PR[91,2] = PR[90,2] + 24.282;
   1:  PR[91,3] = PR[90,3] + 69.970;
   1:L PR[91] R[100]mm/sec CNT100;
   1:  PR[91,1] = PR[90,1] + 48.210;
   1:  PR[91,2] = PR[90,2] + 24.700;
   1:  PR[91,3] = PR[90,3] + 69.981;
   1:L PR[91] R[100]mm/sec CNT100;
   1:  PR[91,1] = PR[90,1] + 46.083;
   1:  PR[91,2] = PR[90,2] + 24.985;
   1:  PR[91,3] = PR[90,3] + 69.988;
   1:L PR[91] R[100]mm/sec CNT100;
   1:  PR[91,1] = PR[90,1] + 42.921;
   1:  PR[91,2] = PR[90,2] + 25.366;
   1:  PR[91,3] = PR[90,3] + 69.996;
   1:L PR[91] R[100]mm/sec CNT100;
   1:  PR[91,1] = PR[90,1] + 39.448;
   1:  PR[91,2] = PR[90,2] + 25.379;
   1:  PR[91,3] = PR[90,3] + 70.007;
   1:L PR[91] R[100]mm/sec CNT100;
   1:  PR[91,1] = PR[90,1] + 37.530;
   1:  PR[91,2] = PR[90,2] + 25.412;
   1:  PR[91,3] = PR[90,3] + 70.020;
   1:L PR[91] R[100]mm/sec CNT100;
   1:  PR[91,1] = PR[90,1] + 36.431;
   1:  PR[91,2] = PR[90,2] + 25.323;
   1:  PR[91,3] = PR[90,3] + 70.027;
   1:L PR[91] R[100]mm/sec CNT100;
   1:  PR[91,1] = PR[90,1] + 32.825;
   1:  PR[91,2] = PR[90,2] + 24.824;
   1:  PR[91,3] = PR[90,3] + 70.031;
   1:L PR[91] R[100]mm/sec CNT100;
   1:  PR[91,1] = PR[90,1] + 29.163;
   1:  PR[91,2] = PR[90,2] + 23.945;
   1:  PR[91,3] = PR[90,3] + 70.044;
   1:L PR[91] R[100]mm/sec CNT100;
   1:  PR[91,1] = PR[90,1] + 27.613;
   1:  PR[91,2] = PR[90,2] + 23.520;
   1:  PR[91,3] = PR[90,3] + 70.058;
   1:L PR[91] R[100]mm/sec CNT100;
   1:  PR[91,1] = PR[90,1] + 25.545;
   1:  PR[91,2] = PR[90,2] + 23.911;
   1:  PR[91,3] = PR[90,3] + 70.064;
   1:L PR[91] R[100]mm/sec CNT100;
   1:  PR[91,1] = PR[90,1] + 22.870;
   1:  PR[91,2] = PR[90,2] + 24.318;
   1:  PR[91,3] = PR[90,3] + 70.071;
   1:L PR[91] R[100]mm/sec CNT100;
   1:  PR[91,1] = PR[90,1] + 21.206;
   1:  PR[91,2] = PR[90,2] + 24.371;
   1:  PR[91,3] = PR[90,3] + 70.081;
   1:L PR[91] R[100]mm/sec CNT100;
   1:  PR[91,1] = PR[90,1] + 17.057;
   1:  PR[91,2] = PR[90,2] + 24.203;
   1:  PR[91,3] = PR[90,3] + 70.087;
   1:L PR[91] R[100]mm/sec CNT100;
   1:  PR[91,1] = PR[90,1] + 15.049;
   1:  PR[91,2] = PR[90,2] + 23.769;
   1:  PR[91,3] = PR[90,3] + 70.102;
   1:L PR[91] R[100]mm/sec CNT100;
   1:  PR[91,1] = PR[90,1] + 11.338;
   1:  PR[91,2] = PR[90,2] + 22.758;
   1:  PR[91,3] = PR[90,3] + 70.110;
   1:L PR[91] R[100]mm/sec CNT100;
   1:  PR[91,1] = PR[90,1] + 7.502;
   1:  PR[91,2] = PR[90,2] + 20.998;
   1:  PR[91,3] = PR[90,3] + 70.124;
   1:L PR[91] R[100]mm/sec CNT100;
   1:  PR[91,1] = PR[90,1] + 5.284;
   1:  PR[91,2] = PR[90,2] + 21.569;
   1:  PR[91,3] = PR[90,3] + 70.139;
   1:L PR[91] R[100]mm/sec CNT100;
   1:  PR[91,1] = PR[90,1] + 0.868;
   1:  PR[91,2] = PR[90,2] + 22.826;
   1:  PR[91,3] = PR[90,3] + 70.147;
   1:L PR[91] R[100]mm/sec CNT100;
   1:  PR[91,1] = PR[90,1] + -0.844;
   1:  PR[91,2] = PR[90,2] + 23.000;
   1:  PR[91,3] = PR[90,3] + 70.164;
   1:L PR[91] R[100]mm/sec CNT100;
   1:  PR[91,1] = PR[90,1] + -5.353;
   1:  PR[91,2] = PR[90,2] + 23.398;
   1:  PR[91,3] = PR[90,3] + 70.170;
   1:L PR[91] R[100]mm/sec CNT100;
   1:  PR[91,1] = PR[90,1] + -9.520;
   1:  PR[91,2] = PR[90,2] + 23.063;
   1:  PR[91,3] = PR[90,3] + 70.187;
   1:L PR[91] R[100]mm/sec CNT100;
   1:  PR[91,1] = PR[90,1] + -11.405;
   1:  PR[91,2] = PR[90,2] + 22.882;
   1:  PR[91,3] = PR[90,3] + 70.202;
   1:L PR[91] R[100]mm/sec CNT100;
   1:  PR[91,1] = PR[90,1] + -13.206;
   1:  PR[91,2] = PR[90,2] + 22.460;
   1:  PR[91,3] = PR[90,3] + 70.209;
   1:L PR[91] R[100]mm/sec CNT100;
   1:  PR[91,1] = PR[90,1] + -16.766;
   1:  PR[91,2] = PR[90,2] + 21.475;
   1:  PR[91,3] = PR[90,3] + 70.216;
   1:L PR[91] R[100]mm/sec CNT100;
   1:  PR[91,1] = PR[90,1] + -17.354;
   1:  PR[91,2] = PR[90,2] + 21.257;
   1:  PR[91,3] = PR[90,3] + 70.229;
   1:L PR[91] R[100]mm/sec CNT100;
   1:  PR[91,1] = PR[90,1] + -20.899;
   1:  PR[91,2] = PR[90,2] + 21.865;
   1:  PR[91,3] = PR[90,3] + 70.231;
   1:L PR[91] R[100]mm/sec CNT100;
   1:  PR[91,1] = PR[90,1] + -21.992;
   1:  PR[91,2] = PR[90,2] + 22.014;
   1:  PR[91,3] = PR[90,3] + 70.244;
   1:L PR[91] R[100]mm/sec CNT100;
   1:  PR[91,1] = PR[90,1] + -26.060;
   1:  PR[91,2] = PR[90,2] + 22.460;
   1:  PR[91,3] = PR[90,3] + 70.248;
   1:L PR[91] R[100]mm/sec CNT100;
   1:  PR[91,1] = PR[90,1] + -29.988;
   1:  PR[91,2] = PR[90,2] + 22.958;
   1:  PR[91,3] = PR[90,3] + 70.263;
   1:L PR[91] R[100]mm/sec CNT100;
   1:  PR[91,1] = PR[90,1] + -34.998;
   1:  PR[91,2] = PR[90,2] + 23.112;
   1:  PR[91,3] = PR[90,3] + 70.278;
   1:L PR[91] R[100]mm/sec CNT100;
   1:  PR[91,1] = PR[90,1] + -38.747;
   1:  PR[91,2] = PR[90,2] + 23.326;
   1:  PR[91,3] = PR[90,3] + 70.296;
   1:L PR[91] R[100]mm/sec CNT100;
   1:  PR[91,1] = PR[90,1] + -46.112;
   1:  PR[91,2] = PR[90,2] + 23.010;
   1:  PR[91,3] = PR[90,3] + 70.310;
   1:L PR[91] R[100]mm/sec CNT100;
   1:  PR[91,1] = PR[90,1] + -50.909;
   1:  PR[91,2] = PR[90,2] + 22.216;
   1:  PR[91,3] = PR[90,3] + 70.336;
   1:L PR[91] R[100]mm/sec CNT100;
   1:  PR[91,1] = PR[90,1] + -55.081;
   1:  PR[91,2] = PR[90,2] + 21.360;
   1:  PR[91,3] = PR[90,3] + 70.354;
   1:L PR[91] R[100]mm/sec CNT100;
   1:  PR[91,1] = PR[90,1] + -55.841;
   1:  PR[91,2] = PR[90,2] + 21.111;
   1:  PR[91,3] = PR[90,3] + 70.370;
   1:L PR[91] R[100]mm/sec CNT100;
   1:  PR[91,1] = PR[90,1] + -57.254;
   1:  PR[91,2] = PR[90,2] + 20.597;
   1:  PR[91,3] = PR[90,3] + 70.373;
   1:L PR[91] R[100]mm/sec CNT100;
   1:  PR[91,1] = PR[90,1] + -61.601;
   1:  PR[91,2] = PR[90,2] + 18.891;
   1:  PR[91,3] = PR[90,3] + 70.378;
   1:L PR[91] R[100]mm/sec CNT100;
   1:  PR[91] = PR[90];
   1:  PR[91,1] = PR[90,1] + -65.707;
   1:  PR[91,2] = PR[90,2] + 15.887;
   1:  PR[91,3] = PR[90,3] + 71.695;
   1:L PR[91] R[100]mm/sec CNT100;
   1:  PR[91,1] = PR[90,1] + -69.794;
   1:  PR[91,2] = PR[90,2] + 12.152;
   1:  PR[91,3] = PR[90,3] + 70.417;
   1:L PR[91] R[100]mm/sec CNT100;
   1:  PR[91,1] = PR[90,1] + -72.717;
   1:  PR[91,2] = PR[90,2] + 8.041;
   1:  PR[91,3] = PR[90,3] + 70.438;
   1:L PR[91] R[100]mm/sec CNT100;
   1:  PR[91,1] = PR[90,1] + -73.488;
   1:  PR[91,2] = PR[90,2] + 6.124;
   1:  PR[91,3] = PR[90,3] + 70.456;
   1:L PR[91] R[100]mm/sec CNT100;
   1:  PR[91,1] = PR[90,1] + -74.386;
   1:  PR[91,2] = PR[90,2] + 3.710;
   1:  PR[91,3] = PR[90,3] + 70.464;
   1:L PR[91] R[100]mm/sec CNT100;
   1:  PR[91,1] = PR[90,1] + -74.450;
   1:  PR[91,2] = PR[90,2] + 3.299;
   1:  PR[91,3] = PR[90,3] + 70.473;
   1:L PR[91] R[100]mm/sec CNT100;
   1:  PR[91,1] = PR[90,1] + -74.948;
   1:  PR[91,2] = PR[90,2] + -0.724;
   1:  PR[91,3] = PR[90,3] + 70.475;
   1:L PR[91] R[100]mm/sec CNT100;
   1:  PR[91,1] = PR[90,1] + -74.870;
   1:  PR[91,2] = PR[90,2] + -1.325;
   1:  PR[91,3] = PR[90,3] + 70.490;
   1:L PR[91] R[100]mm/sec CNT100;
   1:  PR[91,1] = PR[90,1] + -74.374;
   1:  PR[91,2] = PR[90,2] + -3.714;
   1:  PR[91,3] = PR[90,3] + 70.492;
   1:L PR[91] R[100]mm/sec CNT100;
   1:  PR[91,1] = PR[90,1] + -74.163;
   1:  PR[91,2] = PR[90,2] + -5.356;
   1:  PR[91,3] = PR[90,3] + 70.501;
   1:L PR[91] R[100]mm/sec CNT100;
   1:  PR[91,1] = PR[90,1] + -72.349;
   1:  PR[91,2] = PR[90,2] + -9.838;
   1:  PR[91,3] = PR[90,3] + 70.507;
   1:L PR[91] R[100]mm/sec CNT100;
   1:  PR[91,1] = PR[90,1] + -69.351;
   1:  PR[91,2] = PR[90,2] + -14.025;
   1:  PR[91,3] = PR[90,3] + 70.525;
   1:L PR[91] R[100]mm/sec CNT100;
   1:  PR[91,1] = PR[90,1] + -65.242;
   1:  PR[91,2] = PR[90,2] + -17.740;
   1:  PR[91,3] = PR[90,3] + 70.544;
   1:L PR[91] R[100]mm/sec CNT100;
   1:  PR[91,1] = PR[90,1] + -63.201;
   1:  PR[91,2] = PR[90,2] + -18.963;
   1:  PR[91,3] = PR[90,3] + 70.564;
   1:L PR[91] R[100]mm/sec CNT100;
   1:  PR[91,1] = PR[90,1] + -60.149;
   1:  PR[91,2] = PR[90,2] + -20.663;
   1:  PR[91,3] = PR[90,3] + 70.573;
   1:L PR[91] R[100]mm/sec CNT100;
   1:  PR[91,1] = PR[90,1] + -58.545;
   1:  PR[91,2] = PR[90,2] + -21.317;
   1:  PR[91,3] = PR[90,3] + 70.586;
   1:L PR[91] R[100]mm/sec CNT100;
   1:  PR[91,1] = PR[90,1] + -54.554;
   1:  PR[91,2] = PR[90,2] + -22.737;
   1:  PR[91,3] = PR[90,3] + 70.592;
   1:L PR[91] R[100]mm/sec CNT100;
   1:  PR[91,1] = PR[90,1] + -48.807;
   1:  PR[91,2] = PR[90,2] + -24.125;
   1:  PR[91,3] = PR[90,3] + 70.608;
   1:L PR[91] R[100]mm/sec CNT100;
   1:  PR[91,1] = PR[90,1] + -43.240;
   1:  PR[91,2] = PR[90,2] + -24.710;
   1:  PR[91,3] = PR[90,3] + 70.629;
   1:L PR[91] R[100]mm/sec CNT100;
   1:  PR[91,1] = PR[90,1] + -38.259;
   1:  PR[91,2] = PR[90,2] + -25.042;
   1:  PR[91,3] = PR[90,3] + 70.650;
   1:L PR[91] R[100]mm/sec CNT100;
   1:  PR[91,1] = PR[90,1] + -37.657;
   1:  PR[91,2] = PR[90,2] + -25.033;
   1:  PR[91,3] = PR[90,3] + 70.668;
   1:L PR[91] R[100]mm/sec CNT100;
   1:  PR[91,1] = PR[90,1] + -36.948;
   1:  PR[91,2] = PR[90,2] + -24.990;
   1:  PR[91,3] = PR[90,3] + 70.670;
   1:L PR[91] R[100]mm/sec CNT100;
   1:  PR[91,1] = PR[90,1] + -31.514;
   1:  PR[91,2] = PR[90,2] + -24.823;
   1:  PR[91,3] = PR[90,3] + 70.673;
   1:L PR[91] R[100]mm/sec CNT100;
   1:  PR[91,1] = PR[90,1] + -27.586;
   1:  PR[91,2] = PR[90,2] + -24.674;
   1:  PR[91,3] = PR[90,3] + 70.693;
   1:L PR[91] R[100]mm/sec CNT100;
   1:  PR[91,1] = PR[90,1] + -26.716;
   1:  PR[91,2] = PR[90,2] + -24.561;
   1:  PR[91,3] = PR[90,3] + 70.707;
   1:L PR[91] R[100]mm/sec CNT100;
   1:  PR[91,1] = PR[90,1] + -20.035;
   1:  PR[91,2] = PR[90,2] + -23.802;
   1:  PR[91,3] = PR[90,3] + 70.711;
   1:L PR[91] R[100]mm/sec CNT100;
   1:  PR[91,1] = PR[90,1] + -19.700;
   1:  PR[91,2] = PR[90,2] + -23.791;
   1:  PR[91,3] = PR[90,3] + 70.735;
   1:L PR[91] R[100]mm/sec CNT100;
   1:  PR[91,1] = PR[90,1] + -17.905;
   1:  PR[91,2] = PR[90,2] + -23.547;
   1:  PR[91,3] = PR[90,3] + 70.737;
   1:L PR[91] R[100]mm/sec CNT100;
   1:  PR[91,1] = PR[90,1] + -15.931;
   1:  PR[91,2] = PR[90,2] + -23.214;
   1:  PR[91,3] = PR[90,3] + 70.743;
   1:L PR[91] R[100]mm/sec CNT100;
   1:  PR[91,1] = PR[90,1] + -13.554;
   1:  PR[91,2] = PR[90,2] + -23.873;
   1:  PR[91,3] = PR[90,3] + 70.751;
   1:L PR[91] R[100]mm/sec CNT100;
   1:  PR[91,1] = PR[90,1] + -10.713;
   1:  PR[91,2] = PR[90,2] + -24.538;
   1:  PR[91,3] = PR[90,3] + 70.760;
   1:L PR[91] R[100]mm/sec CNT100;
   1:  PR[91,1] = PR[90,1] + -7.719;
   1:  PR[91,2] = PR[90,2] + -24.827;
   1:  PR[91,3] = PR[90,3] + 70.770;
   1:L PR[91] R[100]mm/sec CNT100;
   1:  PR[91,1] = PR[90,1] + -4.615;
   1:  PR[91,2] = PR[90,2] + -25.078;
   1:  PR[91,3] = PR[90,3] + 70.782;
   1:L PR[91] R[100]mm/sec CNT100;
   1:  PR[91,1] = PR[90,1] + 1.671;
   1:  PR[91,2] = PR[90,2] + -24.519;
   1:  PR[91,3] = PR[90,3] + 70.793;
   1:L PR[91] R[100]mm/sec CNT100;
   1:  PR[91,1] = PR[90,1] + 3.293;
   1:  PR[91,2] = PR[90,2] + -24.057;
   1:  PR[91,3] = PR[90,3] + 70.816;
   1:L PR[91] R[100]mm/sec CNT100;
   1:  PR[91,1] = PR[90,1] + 7.849;
   1:  PR[91,2] = PR[90,2] + -22.888;
   1:  PR[91,3] = PR[90,3] + 70.822;
   1:L PR[91] R[100]mm/sec CNT100;
   1:  PR[91,1] = PR[90,1] + 11.205;
   1:  PR[91,2] = PR[90,2] + -24.429;
   1:  PR[91,3] = PR[90,3] + 70.840;
   1:L PR[91] R[100]mm/sec CNT100;
   1:  PR[91,1] = PR[90,1] + 14.352;
   1:  PR[91,2] = PR[90,2] + -25.287;
   1:  PR[91,3] = PR[90,3] + 70.853;
   1:L PR[91] R[100]mm/sec CNT100;
   1:  PR[91,1] = PR[90,1] + 17.021;
   1:  PR[91,2] = PR[90,2] + -25.862;
   1:  PR[91,3] = PR[90,3] + 70.865;
   1:L PR[91] R[100]mm/sec CNT100;
   1:  PR[91,1] = PR[90,1] + 20.601;
   1:  PR[91,2] = PR[90,2] + -26.007;
   1:  PR[91,3] = PR[90,3] + 70.875;
   1:L PR[91] R[100]mm/sec CNT100;
   1:  PR[91,1] = PR[90,1] + 22.920;
   1:  PR[91,2] = PR[90,2] + -25.933;
   1:  PR[91,3] = PR[90,3] + 70.888;
   1:L PR[91] R[100]mm/sec CNT100;
   1:  PR[91,1] = PR[90,1] + 27.084;
   1:  PR[91,2] = PR[90,2] + -25.297;
   1:  PR[91,3] = PR[90,3] + 70.897;
   1:L PR[91] R[100]mm/sec CNT100;
   1:  PR[91,1] = PR[90,1] + 32.347;
   1:  PR[91,2] = PR[90,2] + -26.562;
   1:  PR[91,3] = PR[90,3] + 70.912;
   1:L PR[91] R[100]mm/sec CNT100;
   1:  PR[91,1] = PR[90,1] + 34.823;
   1:  PR[91,2] = PR[90,2] + -26.904;
   1:  PR[91,3] = PR[90,3] + 70.932;
   1:L PR[91] R[100]mm/sec CNT100;
   1:  PR[91,1] = PR[90,1] + 37.170;
   1:  PR[91,2] = PR[90,2] + -27.095;
   1:  PR[91,3] = PR[90,3] + 70.941;
   1:L PR[91] R[100]mm/sec CNT100;
   1:  PR[91,1] = PR[90,1] + 41.084;
   1:  PR[91,2] = PR[90,2] + -27.029;
   1:  PR[91,3] = PR[90,3] + 70.950;
   1:L PR[91] R[100]mm/sec CNT100;
   1:  PR[91,1] = PR[90,1] + 41.965;
   1:  PR[91,2] = PR[90,2] + -27.025;
   1:  PR[91,3] = PR[90,3] + 70.964;
   1:L PR[91] R[100]mm/sec CNT100;
   1:  PR[91,1] = PR[90,1] + 42.741;
   1:  PR[91,2] = PR[90,2] + -26.932;
   1:  PR[91,3] = PR[90,3] + 70.968;
   1:L PR[91] R[100]mm/sec CNT100;
   1:  PR[91,1] = PR[90,1] + 47.420;
   1:  PR[91,2] = PR[90,2] + -26.304;
   1:  PR[91,3] = PR[90,3] + 70.971;
   1:L PR[91] R[100]mm/sec CNT100;
   1:  PR[91,1] = PR[90,1] + 51.088;
   1:  PR[91,2] = PR[90,2] + -25.394;
   1:  PR[91,3] = PR[90,3] + 70.988;
   1:L PR[91] R[100]mm/sec CNT100;
   1:  PR[91,1] = PR[90,1] + 52.146;
   1:  PR[91,2] = PR[90,2] + -25.177;
   1:  PR[91,3] = PR[90,3] + 71.002;
   1:L PR[91] R[100]mm/sec CNT100;
   1:  PR[91,1] = PR[90,1] + 54.710;
   1:  PR[91,2] = PR[90,2] + -24.381;
   1:  PR[91,3] = PR[90,3] + 71.006;
   1:L PR[91] R[100]mm/sec CNT100;
   1:  PR[91,1] = PR[90,1] + 56.598;
   1:  PR[91,2] = PR[90,2] + -23.764;
   1:  PR[91,3] = PR[90,3] + 71.016;
   1:L PR[91] R[100]mm/sec CNT100;
   1:  PR[91,1] = PR[90,1] + 57.363;
   1:  PR[91,2] = PR[90,2] + -23.418;
   1:  PR[91,3] = PR[90,3] + 71.023;
   1:L PR[91] R[100]mm/sec CNT100;
   1:  PR[91,1] = PR[90,1] + 60.603;
   1:  PR[91,2] = PR[90,2] + -21.921;
   1:  PR[91,3] = PR[90,3] + 71.026;
   1:L PR[91] R[100]mm/sec CNT100;
   1:  PR[91,1] = PR[90,1] + 62.414;
   1:  PR[91,2] = PR[90,2] + -20.940;
   1:  PR[91,3] = PR[90,3] + 71.039;
   1:L PR[91] R[100]mm/sec CNT100;
   1:  PR[91,1] = PR[90,1] + 64.886;
   1:  PR[91,2] = PR[90,2] + -19.362;
   1:  PR[91,3] = PR[90,3] + 71.047;
   1:L PR[91] R[100]mm/sec CNT100;
   1:  PR[91,1] = PR[90,1] + 68.573;
   1:  PR[91,2] = PR[90,2] + -16.323;
   1:  PR[91,3] = PR[90,3] + 71.057;
   1:L PR[91] R[100]mm/sec CNT100;
   1:  PR[91,1] = PR[90,1] + 69.278;
   1:  PR[91,2] = PR[90,2] + -15.703;
   1:  PR[91,3] = PR[90,3] + 71.075;
   1:L PR[91] R[100]mm/sec CNT100;
   1:  PR[91,1] = PR[90,1] + 71.943;
   1:  PR[91,2] = PR[90,2] + -12.315;
   1:  PR[91,3] = PR[90,3] + 71.078;
   1:L PR[91] R[100]mm/sec CNT100;
   1:  PR[91,1] = PR[90,1] + 72.860;
   1:  PR[91,2] = PR[90,2] + -11.037;
   1:  PR[91,3] = PR[90,3] + 71.094;
   1:L PR[91] R[100]mm/sec CNT100;
   1:  PR[91,1] = PR[90,1] + 74.909;
   1:  PR[91,2] = PR[90,2] + -5.952;
   1:  PR[91,3] = PR[90,3] + 71.100;
   1:L PR[91] R[100]mm/sec CNT100;
   1:  PR[91,1] = PR[90,1] + 75.021;
   1:  PR[91,2] = PR[90,2] + -5.106;
   1:  PR[91,3] = PR[90,3] + 71.120;
   1:L PR[91] R[100]mm/sec CNT100;
   1:  PR[91,1] = PR[90,1] + 75.710;
   1:  PR[91,2] = PR[90,2] + -0.815;
   1:  PR[91,3] = PR[90,3] + 71.123;
   1:L PR[91] R[100]mm/sec CNT100;
   1:  PR[91,1] = PR[90,1] + 75.480;
   1:  PR[91,2] = PR[90,2] + 0.111;
   1:  PR[91,3] = PR[90,3] + 71.139;
   1:L PR[91] R[100]mm/sec CNT100;
   1:  PR[91,1] = PR[90,1] + 74.909;
   1:  PR[91,2] = PR[90,2] + 4.493;
   1:  PR[91,3] = PR[90,3] + 71.143;
   1:L PR[91] R[100]mm/sec CNT100;
   1:  PR[91,1] = PR[90,1] + 72.862;
   1:  PR[91,2] = PR[90,2] + 9.573;
   1:  PR[91,3] = PR[90,3] + 71.159;
   1:L PR[91] R[100]mm/sec CNT100;
   1:  PR[91,1] = PR[90,1] + 71.941;
   1:  PR[91,2] = PR[90,2] + 10.859;
   1:  PR[91,3] = PR[90,3] + 71.179;
   1:L PR[91] R[100]mm/sec CNT100;
   1:  PR[91,1] = PR[90,1] + 69.608;
   1:  PR[91,2] = PR[90,2] + 13.845;
   1:  PR[91,3] = PR[90,3] + 71.185;
   1:L PR[91] R[100]mm/sec CNT100;
   1:  PR[91,1] = PR[90,1] + 69.298;
   1:  PR[91,2] = PR[90,2] + 14.226;
   1:  PR[91,3] = PR[90,3] + 71.199;
   1:L PR[91] R[100]mm/sec CNT100;
   1:  PR[91,1] = PR[90,1] + 68.582;
   1:  PR[91,2] = PR[90,2] + 14.856;
   1:  PR[91,3] = PR[90,3] + 71.201;
   1:L PR[91] R[100]mm/sec CNT100;
   1:  PR[91,1] = PR[90,1] + 64.894;
   1:  PR[91,2] = PR[90,2] + 17.899;
   1:  PR[91,3] = PR[90,3] + 71.204;
   1:L PR[91] R[100]mm/sec CNT100;
   1:  PR[91,1] = PR[90,1] + 62.420;
   1:  PR[91,2] = PR[90,2] + 19.477;
   1:  PR[91,3] = PR[90,3] + 71.222;
   1:L PR[91] R[100]mm/sec CNT100;
   1:  PR[91,1] = PR[90,1] + 60.608;
   1:  PR[91,2] = PR[90,2] + 20.459;
   1:  PR[91,3] = PR[90,3] + 71.233;
   1:L PR[91] R[100]mm/sec CNT100;
   1:  PR[91,1] = PR[90,1] + 56.591;
   1:  PR[91,2] = PR[90,2] + 22.307;
   1:  PR[91,3] = PR[90,3] + 71.240;
   1:L PR[91] R[100]mm/sec CNT100;
   1:  PR[91,1] = PR[90,1] + 54.711;
   1:  PR[91,2] = PR[90,2] + 22.922;
   1:  PR[91,3] = PR[90,3] + 71.256;
   1:L PR[91] R[100]mm/sec CNT100;
   1:  PR[91,1] = PR[90,1] + 52.146;
   1:  PR[91,2] = PR[90,2] + 23.718;
   1:  PR[91,3] = PR[90,3] + 71.264;
   1:L PR[91] R[100]mm/sec CNT100;
   1:  PR[91,1] = PR[90,1] + 51.088;
   1:  PR[91,2] = PR[90,2] + 23.935;
   1:  PR[91,3] = PR[90,3] + 71.274;
   1:L PR[91] R[100]mm/sec CNT100;
   1:  PR[91,1] = PR[90,1] + 47.420;
   1:  PR[91,2] = PR[90,2] + 24.845;
   1:  PR[91,3] = PR[90,3] + 71.278;
   1:L PR[91] R[100]mm/sec CNT100;
   1:  PR[91,1] = PR[90,1] + 42.741;
   1:  PR[91,2] = PR[90,2] + 25.473;
   1:  PR[91,3] = PR[90,3] + 71.291;
   1:L PR[91] R[100]mm/sec CNT100;
   1:  PR[91,1] = PR[90,1] + 41.965;
   1:  PR[91,2] = PR[90,2] + 25.566;
   1:  PR[91,3] = PR[90,3] + 71.309;
   1:L PR[91] R[100]mm/sec CNT100;
   1:  PR[91,1] = PR[90,1] + 41.084;
   1:  PR[91,2] = PR[90,2] + 25.570;
   1:  PR[91,3] = PR[90,3] + 71.312;
   1:L PR[91] R[100]mm/sec CNT100;
   1:  PR[91,1] = PR[90,1] + 37.170;
   1:  PR[91,2] = PR[90,2] + 25.636;
   1:  PR[91,3] = PR[90,3] + 71.315;
   1:L PR[91] R[100]mm/sec CNT100;
   1:  PR[91,1] = PR[90,1] + 34.823;
   1:  PR[91,2] = PR[90,2] + 25.445;
   1:  PR[91,3] = PR[90,3] + 71.329;
   1:L PR[91] R[100]mm/sec CNT100;
   1:  PR[91,1] = PR[90,1] + 32.347;
   1:  PR[91,2] = PR[90,2] + 25.103;
   1:  PR[91,3] = PR[90,3] + 71.338;
   1:L PR[91] R[100]mm/sec CNT100;
   1:  PR[91,1] = PR[90,1] + 27.084;
   1:  PR[91,2] = PR[90,2] + 23.838;
   1:  PR[91,3] = PR[90,3] + 71.347;
   1:L PR[91] R[100]mm/sec CNT100;
   1:  PR[91,1] = PR[90,1] + 22.919;
   1:  PR[91,2] = PR[90,2] + 24.474;
   1:  PR[91,3] = PR[90,3] + 71.367;
   1:L PR[91] R[100]mm/sec CNT100;
   1:  PR[91,1] = PR[90,1] + 20.600;
   1:  PR[91,2] = PR[90,2] + 24.549;
   1:  PR[91,3] = PR[90,3] + 71.382;
   1:L PR[91] R[100]mm/sec CNT100;
   1:  PR[91,1] = PR[90,1] + 17.020;
   1:  PR[91,2] = PR[90,2] + 24.403;
   1:  PR[91,3] = PR[90,3] + 71.391;
   1:L PR[91] R[100]mm/sec CNT100;
   1:  PR[91,1] = PR[90,1] + 14.351;
   1:  PR[91,2] = PR[90,2] + 23.828;
   1:  PR[91,3] = PR[90,3] + 71.404;
   1:L PR[91] R[100]mm/sec CNT100;
   1:  PR[91,1] = PR[90,1] + 11.204;
   1:  PR[91,2] = PR[90,2] + 22.970;
   1:  PR[91,3] = PR[90,3] + 71.414;
   1:L PR[91] R[100]mm/sec CNT100;
   1:  PR[91,1] = PR[90,1] + 7.848;
   1:  PR[91,2] = PR[90,2] + 21.430;
   1:  PR[91,3] = PR[90,3] + 71.426;
   1:L PR[91] R[100]mm/sec CNT100;
   1:  PR[91,1] = PR[90,1] + 3.303;
   1:  PR[91,2] = PR[90,2] + 22.600;
   1:  PR[91,3] = PR[90,3] + 71.440;
   1:L PR[91] R[100]mm/sec CNT100;
   1:  PR[91,1] = PR[90,1] + 1.714;
   1:  PR[91,2] = PR[90,2] + 23.052;
   1:  PR[91,3] = PR[90,3] + 71.457;
   1:L PR[91] R[100]mm/sec CNT100;
   1:  PR[91,1] = PR[90,1] + -4.595;
   1:  PR[91,2] = PR[90,2] + 23.619;
   1:  PR[91,3] = PR[90,3] + 71.463;
   1:L PR[91] R[100]mm/sec CNT100;
   1:  PR[91,1] = PR[90,1] + -7.696;
   1:  PR[91,2] = PR[90,2] + 23.369;
   1:  PR[91,3] = PR[90,3] + 71.486;
   1:L PR[91] R[100]mm/sec CNT100;
   1:  PR[91,1] = PR[90,1] + -10.709;
   1:  PR[91,2] = PR[90,2] + 23.080;
   1:  PR[91,3] = PR[90,3] + 71.498;
   1:L PR[91] R[100]mm/sec CNT100;
   1:  PR[91,1] = PR[90,1] + -13.600;
   1:  PR[91,2] = PR[90,2] + 22.402;
   1:  PR[91,3] = PR[90,3] + 71.509;
   1:L PR[91] R[100]mm/sec CNT100;
   1:  PR[91,1] = PR[90,1] + -15.931;
   1:  PR[91,2] = PR[90,2] + 21.755;
   1:  PR[91,3] = PR[90,3] + 71.520;
   1:L PR[91] R[100]mm/sec CNT100;
   1:  PR[91,1] = PR[90,1] + -17.870;
   1:  PR[91,2] = PR[90,2] + 22.083;
   1:  PR[91,3] = PR[90,3] + 71.529;
   1:L PR[91] R[100]mm/sec CNT100;
   1:  PR[91,1] = PR[90,1] + -19.775;
   1:  PR[91,2] = PR[90,2] + 22.343;
   1:  PR[91,3] = PR[90,3] + 71.536;
   1:L PR[91] R[100]mm/sec CNT100;
   1:  PR[91,1] = PR[90,1] + -26.709;
   1:  PR[91,2] = PR[90,2] + 23.102;
   1:  PR[91,3] = PR[90,3] + 71.543;
   1:L PR[91] R[100]mm/sec CNT100;
   1:  PR[91,1] = PR[90,1] + -27.634;
   1:  PR[91,2] = PR[90,2] + 23.219;
   1:  PR[91,3] = PR[90,3] + 71.569;
   1:L PR[91] R[100]mm/sec CNT100;
   1:  PR[91,1] = PR[90,1] + -35.837;
   1:  PR[91,2] = PR[90,2] + 23.471;
   1:  PR[91,3] = PR[90,3] + 71.572;
   1:L PR[91] R[100]mm/sec CNT100;
   1:  PR[91,1] = PR[90,1] + -37.663;
   1:  PR[91,2] = PR[90,2] + 23.575;
   1:  PR[91,3] = PR[90,3] + 71.602;
   1:L PR[91] R[100]mm/sec CNT100;
   1:  PR[91,1] = PR[90,1] + -41.865;
   1:  PR[91,2] = PR[90,2] + 23.392;
   1:  PR[91,3] = PR[90,3] + 71.609;
   1:L PR[91] R[100]mm/sec CNT100;
   1:  PR[91,1] = PR[90,1] + -44.716;
   1:  PR[91,2] = PR[90,2] + 23.204;
   1:  PR[91,3] = PR[90,3] + 71.624;
   1:L PR[91] R[100]mm/sec CNT100;
   1:  PR[91,1] = PR[90,1] + -50.383;
   1:  PR[91,2] = PR[90,2] + 22.257;
   1:  PR[91,3] = PR[90,3] + 71.635;
   1:L PR[91] R[100]mm/sec CNT100;
   1:  PR[91,1] = PR[90,1] + -53.393;
   1:  PR[91,2] = PR[90,2] + 21.640;
   1:  PR[91,3] = PR[90,3] + 71.656;
   1:L PR[91] R[100]mm/sec CNT100;
   1:  PR[91,1] = PR[90,1] + -55.296;
   1:  PR[91,2] = PR[90,2] + 21.017;
   1:  PR[91,3] = PR[90,3] + 71.667;
   1:L PR[91] R[100]mm/sec CNT100;
   1:  PR[91,1] = PR[90,1] + -58.574;
   1:  PR[91,2] = PR[90,2] + 19.824;
   1:  PR[91,3] = PR[90,3] + 71.675;
   1:L PR[91] R[100]mm/sec CNT100;
   1:  PR[91,1] = PR[90,1] + -60.495;
   1:  PR[91,2] = PR[90,2] + 19.070;
   1:  PR[91,3] = PR[90,3] + 71.687;
   1:L PR[91] R[100]mm/sec CNT100;
   1:  PR[91] = PR[90];
   1:  PR[91,1] = PR[90,1] + -64.658;
   1:  PR[91,2] = PR[90,2] + 16.036;
   1:  PR[91,3] = PR[90,3] + 72.995;
   1:L PR[91] R[100]mm/sec CNT100;
   1:  PR[91,1] = PR[90,1] + -66.807;
   1:  PR[91,2] = PR[90,2] + 14.084;
   1:  PR[91,3] = PR[90,3] + 71.717;
   1:L PR[91] R[100]mm/sec CNT100;
   1:  PR[91,1] = PR[90,1] + -68.784;
   1:  PR[91,2] = PR[90,2] + 12.271;
   1:  PR[91,3] = PR[90,3] + 71.728;
   1:L PR[91] R[100]mm/sec CNT100;
   1:  PR[91,1] = PR[90,1] + -71.738;
   1:  PR[91,2] = PR[90,2] + 8.120;
   1:  PR[91,3] = PR[90,3] + 71.738;
   1:L PR[91] R[100]mm/sec CNT100;
   1:  PR[91,1] = PR[90,1] + -73.499;
   1:  PR[91,2] = PR[90,2] + 3.745;
   1:  PR[91,3] = PR[90,3] + 71.757;
   1:L PR[91] R[100]mm/sec CNT100;
   1:  PR[91,1] = PR[90,1] + -74.080;
   1:  PR[91,2] = PR[90,2] + -0.689;
   1:  PR[91,3] = PR[90,3] + 71.774;
   1:L PR[91] R[100]mm/sec CNT100;
   1:  PR[91,1] = PR[90,1] + -73.575;
   1:  PR[91,2] = PR[90,2] + -3.117;
   1:  PR[91,3] = PR[90,3] + 71.791;
   1:L PR[91] R[100]mm/sec CNT100;
   1:  PR[91,1] = PR[90,1] + -73.284;
   1:  PR[91,2] = PR[90,2] + -5.386;
   1:  PR[91,3] = PR[90,3] + 71.800;
   1:L PR[91] R[100]mm/sec CNT100;
   1:  PR[91,1] = PR[90,1] + -72.278;
   1:  PR[91,2] = PR[90,2] + -7.892;
   1:  PR[91,3] = PR[90,3] + 71.808;
   1:L PR[91] R[100]mm/sec CNT100;
   1:  PR[91,1] = PR[90,1] + -71.464;
   1:  PR[91,2] = PR[90,2] + -9.892;
   1:  PR[91,3] = PR[90,3] + 71.818;
   1:L PR[91] R[100]mm/sec CNT100;
   1:  PR[91,1] = PR[90,1] + -68.451;
   1:  PR[91,2] = PR[90,2] + -14.108;
   1:  PR[91,3] = PR[90,3] + 71.826;
   1:L PR[91] R[100]mm/sec CNT100;
   1:  PR[91,1] = PR[90,1] + -64.359;
   1:  PR[91,2] = PR[90,2] + -17.817;
   1:  PR[91,3] = PR[90,3] + 71.846;
   1:L PR[91] R[100]mm/sec CNT100;
   1:  PR[91,1] = PR[90,1] + -59.208;
   1:  PR[91,2] = PR[90,2] + -20.687;
   1:  PR[91,3] = PR[90,3] + 71.866;
   1:L PR[91] R[100]mm/sec CNT100;
   1:  PR[91,1] = PR[90,1] + -56.302;
   1:  PR[91,2] = PR[90,2] + -21.871;
   1:  PR[91,3] = PR[90,3] + 71.888;
   1:L PR[91] R[100]mm/sec CNT100;
   1:  PR[91,1] = PR[90,1] + -53.674;
   1:  PR[91,2] = PR[90,2] + -22.806;
   1:  PR[91,3] = PR[90,3] + 71.900;
   1:L PR[91] R[100]mm/sec CNT100;
   1:  PR[91,1] = PR[90,1] + -49.742;
   1:  PR[91,2] = PR[90,2] + -23.757;
   1:  PR[91,3] = PR[90,3] + 71.910;
   1:L PR[91] R[100]mm/sec CNT100;
   1:  PR[91,1] = PR[90,1] + -47.986;
   1:  PR[91,2] = PR[90,2] + -24.162;
   1:  PR[91,3] = PR[90,3] + 71.925;
   1:L PR[91] R[100]mm/sec CNT100;
   1:  PR[91,1] = PR[90,1] + -46.736;
   1:  PR[91,2] = PR[90,2] + -24.408;
   1:  PR[91,3] = PR[90,3] + 71.932;
   1:L PR[91] R[100]mm/sec CNT100;
   1:  PR[91,1] = PR[90,1] + -42.499;
   1:  PR[91,2] = PR[90,2] + -24.853;
   1:  PR[91,3] = PR[90,3] + 71.937;
   1:L PR[91] R[100]mm/sec CNT100;
   1:  PR[91,1] = PR[90,1] + -37.572;
   1:  PR[91,2] = PR[90,2] + -25.182;
   1:  PR[91,3] = PR[90,3] + 71.952;
   1:L PR[91] R[100]mm/sec CNT100;
   1:  PR[91,1] = PR[90,1] + -36.488;
   1:  PR[91,2] = PR[90,2] + -25.268;
   1:  PR[91,3] = PR[90,3] + 71.971;
   1:L PR[91] R[100]mm/sec CNT100;
   1:  PR[91,1] = PR[90,1] + -35.528;
   1:  PR[91,2] = PR[90,2] + -25.297;
   1:  PR[91,3] = PR[90,3] + 71.975;
   1:L PR[91] R[100]mm/sec CNT100;
   1:  PR[91,1] = PR[90,1] + -30.632;
   1:  PR[91,2] = PR[90,2] + -25.146;
   1:  PR[91,3] = PR[90,3] + 71.978;
   1:L PR[91] R[100]mm/sec CNT100;
   1:  PR[91,1] = PR[90,1] + -24.961;
   1:  PR[91,2] = PR[90,2] + -24.930;
   1:  PR[91,3] = PR[90,3] + 71.996;
   1:L PR[91] R[100]mm/sec CNT100;
   1:  PR[91,1] = PR[90,1] + -17.966;
   1:  PR[91,2] = PR[90,2] + -24.135;
   1:  PR[91,3] = PR[90,3] + 72.017;
   1:L PR[91] R[100]mm/sec CNT100;
   1:  PR[91,1] = PR[90,1] + -17.484;
   1:  PR[91,2] = PR[90,2] + -24.120;
   1:  PR[91,3] = PR[90,3] + 72.044;
   1:L PR[91] R[100]mm/sec CNT100;
   1:  PR[91,1] = PR[90,1] + -14.422;
   1:  PR[91,2] = PR[90,2] + -23.701;
   1:  PR[91,3] = PR[90,3] + 72.045;
   1:L PR[91] R[100]mm/sec CNT100;
   1:  PR[91,1] = PR[90,1] + -10.015;
   1:  PR[91,2] = PR[90,2] + -24.736;
   1:  PR[91,3] = PR[90,3] + 72.057;
   1:L PR[91] R[100]mm/sec CNT100;
   1:  PR[91,1] = PR[90,1] + -5.899;
   1:  PR[91,2] = PR[90,2] + -25.133;
   1:  PR[91,3] = PR[90,3] + 72.074;
   1:L PR[91] R[100]mm/sec CNT100;
   1:  PR[91,1] = PR[90,1] + -3.854;
   1:  PR[91,2] = PR[90,2] + -25.298;
   1:  PR[91,3] = PR[90,3] + 72.089;
   1:L PR[91] R[100]mm/sec CNT100;
   1:  PR[91,1] = PR[90,1] + 2.663;
   1:  PR[91,2] = PR[90,2] + -24.737;
   1:  PR[91,3] = PR[90,3] + 72.097;
   1:L PR[91] R[100]mm/sec CNT100;
   1:  PR[91,1] = PR[90,1] + 8.196;
   1:  PR[91,2] = PR[90,2] + -23.321;
   1:  PR[91,3] = PR[90,3] + 72.121;
   1:L PR[91] R[100]mm/sec CNT100;
   1:  PR[91,1] = PR[90,1] + 11.071;
   1:  PR[91,2] = PR[90,2] + -24.641;
   1:  PR[91,3] = PR[90,3] + 72.142;
   1:L PR[91] R[100]mm/sec CNT100;
   1:  PR[91,1] = PR[90,1] + 13.655;
   1:  PR[91,2] = PR[90,2] + -25.345;
   1:  PR[91,3] = PR[90,3] + 72.154;
   1:L PR[91] R[100]mm/sec CNT100;
   1:  PR[91,1] = PR[90,1] + 16.983;
   1:  PR[91,2] = PR[90,2] + -26.063;
   1:  PR[91,3] = PR[90,3] + 72.164;
   1:L PR[91] R[100]mm/sec CNT100;
   1:  PR[91,1] = PR[90,1] + 19.995;
   1:  PR[91,2] = PR[90,2] + -26.185;
   1:  PR[91,3] = PR[90,3] + 72.176;
   1:L PR[91] R[100]mm/sec CNT100;
   1:  PR[91,1] = PR[90,1] + 22.970;
   1:  PR[91,2] = PR[90,2] + -26.089;
   1:  PR[91,3] = PR[90,3] + 72.188;
   1:L PR[91] R[100]mm/sec CNT100;
   1:  PR[91,1] = PR[90,1] + 26.634;
   1:  PR[91,2] = PR[90,2] + -25.533;
   1:  PR[91,3] = PR[90,3] + 72.199;
   1:L PR[91] R[100]mm/sec CNT100;
   1:  PR[91,1] = PR[90,1] + 29.088;
   1:  PR[91,2] = PR[90,2] + -26.173;
   1:  PR[91,3] = PR[90,3] + 72.212;
   1:L PR[91] R[100]mm/sec CNT100;
   1:  PR[91,1] = PR[90,1] + 31.868;
   1:  PR[91,2] = PR[90,2] + -26.840;
   1:  PR[91,3] = PR[90,3] + 72.222;
   1:L PR[91] R[100]mm/sec CNT100;
   1:  PR[91,1] = PR[90,1] + 33.215;
   1:  PR[91,2] = PR[90,2] + -27.027;
   1:  PR[91,3] = PR[90,3] + 72.232;
   1:L PR[91] R[100]mm/sec CNT100;
   1:  PR[91,1] = PR[90,1] + 36.811;
   1:  PR[91,2] = PR[90,2] + -27.319;
   1:  PR[91,3] = PR[90,3] + 72.237;
   1:L PR[91] R[100]mm/sec CNT100;
   1:  PR[91,1] = PR[90,1] + 40.668;
   1:  PR[91,2] = PR[90,2] + -27.254;
   1:  PR[91,3] = PR[90,3] + 72.251;
   1:L PR[91] R[100]mm/sec CNT100;
   1:  PR[91,1] = PR[90,1] + 41.328;
   1:  PR[91,2] = PR[90,2] + -27.203;
   1:  PR[91,3] = PR[90,3] + 72.265;
   1:L PR[91] R[100]mm/sec CNT100;
   1:  PR[91,1] = PR[90,1] + 42.439;
   1:  PR[91,2] = PR[90,2] + -27.011;
   1:  PR[91,3] = PR[90,3] + 72.268;
   1:L PR[91] R[100]mm/sec CNT100;
   1:  PR[91,1] = PR[90,1] + 46.630;
   1:  PR[91,2] = PR[90,2] + -26.449;
   1:  PR[91,3] = PR[90,3] + 72.272;
   1:L PR[91] R[100]mm/sec CNT100;
   1:  PR[91,1] = PR[90,1] + 50.455;
   1:  PR[91,2] = PR[90,2] + -25.500;
   1:  PR[91,3] = PR[90,3] + 72.288;
   1:L PR[91] R[100]mm/sec CNT100;
   1:  PR[91,1] = PR[90,1] + 51.336;
   1:  PR[91,2] = PR[90,2] + -25.262;
   1:  PR[91,3] = PR[90,3] + 72.302;
   1:L PR[91] R[100]mm/sec CNT100;
   1:  PR[91,1] = PR[90,1] + 52.051;
   1:  PR[91,2] = PR[90,2] + -24.984;
   1:  PR[91,3] = PR[90,3] + 72.306;
   1:L PR[91] R[100]mm/sec CNT100;
   1:  PR[91,1] = PR[90,1] + 55.819;
   1:  PR[91,2] = PR[90,2] + -23.752;
   1:  PR[91,3] = PR[90,3] + 72.308;
   1:L PR[91] R[100]mm/sec CNT100;
   1:  PR[91,1] = PR[90,1] + 60.017;
   1:  PR[91,2] = PR[90,2] + -21.841;
   1:  PR[91,3] = PR[90,3] + 72.323;
   1:L PR[91] R[100]mm/sec CNT100;
   1:  PR[91,1] = PR[90,1] + 60.781;
   1:  PR[91,2] = PR[90,2] + -21.428;
   1:  PR[91,3] = PR[90,3] + 72.340;
   1:L PR[91] R[100]mm/sec CNT100;
   1:  PR[91,1] = PR[90,1] + 64.071;
   1:  PR[91,2] = PR[90,2] + -19.328;
   1:  PR[91,3] = PR[90,3] + 72.343;
   1:L PR[91] R[100]mm/sec CNT100;
   1:  PR[91,1] = PR[90,1] + 66.786;
   1:  PR[91,2] = PR[90,2] + -17.090;
   1:  PR[91,3] = PR[90,3] + 72.358;
   1:L PR[91] R[100]mm/sec CNT100;
   1:  PR[91,1] = PR[90,1] + 68.269;
   1:  PR[91,2] = PR[90,2] + -15.785;
   1:  PR[91,3] = PR[90,3] + 72.371;
   1:L PR[91] R[100]mm/sec CNT100;
   1:  PR[91,1] = PR[90,1] + 71.977;
   1:  PR[91,2] = PR[90,2] + -11.080;
   1:  PR[91,3] = PR[90,3] + 72.378;
   1:L PR[91] R[100]mm/sec CNT100;
   1:  PR[91,1] = PR[90,1] + 72.022;
   1:  PR[91,2] = PR[90,2] + -10.999;
   1:  PR[91,3] = PR[90,3] + 72.401;
   1:L PR[91] R[100]mm/sec CNT100;
   1:  PR[91,1] = PR[90,1] + 73.204;
   1:  PR[91,2] = PR[90,2] + -8.301;
   1:L PR[91] R[100]mm/sec CNT100;
   1:  PR[91,1] = PR[90,1] + 74.139;
   1:  PR[91,2] = PR[90,2] + -5.981;
   1:  PR[91,3] = PR[90,3] + 72.412;
   1:L PR[91] R[100]mm/sec CNT100;
   1:  PR[91,1] = PR[90,1] + 74.388;
   1:  PR[91,2] = PR[90,2] + -4.382;
   1:  PR[91,3] = PR[90,3] + 72.421;
   1:L PR[91] R[100]mm/sec CNT100;
   1:  PR[91,1] = PR[90,1] + 74.867;
   1:  PR[91,2] = PR[90,2] + -0.844;
   1:  PR[91,3] = PR[90,3] + 72.427;
   1:L PR[91] R[100]mm/sec CNT100;
   1:  PR[91,1] = PR[90,1] + 74.796;
   1:  PR[91,2] = PR[90,2] + -0.562;
   1:  PR[91,3] = PR[90,3] + 72.440;
   1:L PR[91] R[100]mm/sec CNT100;
   1:  PR[91,1] = PR[90,1] + 74.131;
   1:  PR[91,2] = PR[90,2] + 4.543;
   1:  PR[91,3] = PR[90,3] + 72.441;
   1:L PR[91] R[100]mm/sec CNT100;
   1:  PR[91,1] = PR[90,1] + 73.204;
   1:  PR[91,2] = PR[90,2] + 6.843;
   1:  PR[91,3] = PR[90,3] + 72.461;
   1:L PR[91] R[100]mm/sec CNT100;
   1:  PR[91,1] = PR[90,1] + 72.026;
   1:  PR[91,2] = PR[90,2] + 9.535;
   1:  PR[91,3] = PR[90,3] + 72.470;
   1:L PR[91] R[100]mm/sec CNT100;
   1:  PR[91,1] = PR[90,1] + 71.979;
   1:  PR[91,2] = PR[90,2] + 9.618;
   1:  PR[91,3] = PR[90,3] + 72.481;
   1:L PR[91] R[100]mm/sec CNT100;
   1:  PR[91,1] = PR[90,1] + 68.980;
   1:  PR[91,2] = PR[90,2] + 13.457;
   1:L PR[91] R[100]mm/sec CNT100;
   1:  PR[91,1] = PR[90,1] + 68.287;
   1:  PR[91,2] = PR[90,2] + 14.310;
   1:  PR[91,3] = PR[90,3] + 72.499;
   1:L PR[91] R[100]mm/sec CNT100;
   1:  PR[91,1] = PR[90,1] + 66.792;
   1:  PR[91,2] = PR[90,2] + 15.625;
   1:  PR[91,3] = PR[90,3] + 72.503;
   1:L PR[91] R[100]mm/sec CNT100;
   1:  PR[91,1] = PR[90,1] + 64.076;
   1:  PR[91,2] = PR[90,2] + 17.866;
   1:  PR[91,3] = PR[90,3] + 72.511;
   1:L PR[91] R[100]mm/sec CNT100;
   1:  PR[91,1] = PR[90,1] + 60.784;
   1:  PR[91,2] = PR[90,2] + 19.967;
   1:  PR[91,3] = PR[90,3] + 72.524;
   1:L PR[91] R[100]mm/sec CNT100;
   1:  PR[91,1] = PR[90,1] + 60.019;
   1:  PR[91,2] = PR[90,2] + 20.382;
   1:  PR[91,3] = PR[90,3] + 72.538;
   1:L PR[91] R[100]mm/sec CNT100;
   1:  PR[91,1] = PR[90,1] + 55.819;
   1:  PR[91,2] = PR[90,2] + 22.294;
   1:  PR[91,3] = PR[90,3] + 72.541;
   1:L PR[91] R[100]mm/sec CNT100;
   1:  PR[91,1] = PR[90,1] + 52.051;
   1:  PR[91,2] = PR[90,2] + 23.525;
   1:  PR[91,3] = PR[90,3] + 72.558;
   1:L PR[91] R[100]mm/sec CNT100;
   1:  PR[91,1] = PR[90,1] + 51.336;
   1:  PR[91,2] = PR[90,2] + 23.803;
   1:  PR[91,3] = PR[90,3] + 72.573;
   1:L PR[91] R[100]mm/sec CNT100;
   1:  PR[91,1] = PR[90,1] + 50.455;
   1:  PR[91,2] = PR[90,2] + 24.041;
   1:  PR[91,3] = PR[90,3] + 72.576;
   1:L PR[91] R[100]mm/sec CNT100;
   1:  PR[91,1] = PR[90,1] + 46.630;
   1:  PR[91,2] = PR[90,2] + 24.990;
   1:  PR[91,3] = PR[90,3] + 72.579;
   1:L PR[91] R[100]mm/sec CNT100;
   1:  PR[91,1] = PR[90,1] + 42.439;
   1:  PR[91,2] = PR[90,2] + 25.553;
   1:  PR[91,3] = PR[90,3] + 72.594;
   1:L PR[91] R[100]mm/sec CNT100;
   1:  PR[91,1] = PR[90,1] + 41.328;
   1:  PR[91,2] = PR[90,2] + 25.744;
   1:  PR[91,3] = PR[90,3] + 72.610;
   1:L PR[91] R[100]mm/sec CNT100;
   1:  PR[91,1] = PR[90,1] + 40.668;
   1:  PR[91,2] = PR[90,2] + 25.795;
   1:  PR[91,3] = PR[90,3] + 72.614;
   1:L PR[91] R[100]mm/sec CNT100;
   1:  PR[91,1] = PR[90,1] + 36.811;
   1:  PR[91,2] = PR[90,2] + 25.860;
   1:  PR[91,3] = PR[90,3] + 72.616;
   1:L PR[91] R[100]mm/sec CNT100;
   1:  PR[91,1] = PR[90,1] + 33.215;
   1:  PR[91,2] = PR[90,2] + 25.568;
   1:  PR[91,3] = PR[90,3] + 72.631;
   1:L PR[91] R[100]mm/sec CNT100;
   1:  PR[91,1] = PR[90,1] + 31.868;
   1:  PR[91,2] = PR[90,2] + 25.382;
   1:  PR[91,3] = PR[90,3] + 72.644;
   1:L PR[91] R[100]mm/sec CNT100;
   1:  PR[91,1] = PR[90,1] + 29.088;
   1:  PR[91,2] = PR[90,2] + 24.714;
   1:  PR[91,3] = PR[90,3] + 72.649;
   1:L PR[91] R[100]mm/sec CNT100;
   1:  PR[91,1] = PR[90,1] + 26.634;
   1:  PR[91,2] = PR[90,2] + 24.074;
   1:  PR[91,3] = PR[90,3] + 72.660;
   1:L PR[91] R[100]mm/sec CNT100;
   1:  PR[91,1] = PR[90,1] + 22.970;
   1:  PR[91,2] = PR[90,2] + 24.630;
   1:  PR[91,3] = PR[90,3] + 72.669;
   1:L PR[91] R[100]mm/sec CNT100;
   1:  PR[91,1] = PR[90,1] + 19.995;
   1:  PR[91,2] = PR[90,2] + 24.726;
   1:  PR[91,3] = PR[90,3] + 72.683;
   1:L PR[91] R[100]mm/sec CNT100;
   1:  PR[91,1] = PR[90,1] + 16.982;
   1:  PR[91,2] = PR[90,2] + 24.604;
   1:  PR[91,3] = PR[90,3] + 72.694;
   1:L PR[91] R[100]mm/sec CNT100;
   1:  PR[91,1] = PR[90,1] + 13.654;
   1:  PR[91,2] = PR[90,2] + 23.886;
   1:  PR[91,3] = PR[90,3] + 72.705;
   1:L PR[91] R[100]mm/sec CNT100;
   1:  PR[91,1] = PR[90,1] + 11.070;
   1:  PR[91,2] = PR[90,2] + 23.182;
   1:  PR[91,3] = PR[90,3] + 72.718;
   1:L PR[91] R[100]mm/sec CNT100;
   1:  PR[91,1] = PR[90,1] + 8.194;
   1:  PR[91,2] = PR[90,2] + 21.862;
   1:  PR[91,3] = PR[90,3] + 72.728;
   1:L PR[91] R[100]mm/sec CNT100;
   1:  PR[91,1] = PR[90,1] + 2.710;
   1:  PR[91,2] = PR[90,2] + 23.270;
   1:  PR[91,3] = PR[90,3] + 72.739;
   1:L PR[91] R[100]mm/sec CNT100;
   1:  PR[91,1] = PR[90,1] + -3.833;
   1:  PR[91,2] = PR[90,2] + 23.839;
   1:  PR[91,3] = PR[90,3] + 72.760;
   1:L PR[91] R[100]mm/sec CNT100;
   1:  PR[91,1] = PR[90,1] + -5.873;
   1:  PR[91,2] = PR[90,2] + 23.675;
   1:  PR[91,3] = PR[90,3] + 72.785;
   1:L PR[91] R[100]mm/sec CNT100;
   1:  PR[91,1] = PR[90,1] + -10.012;
   1:  PR[91,2] = PR[90,2] + 23.278;
   1:  PR[91,3] = PR[90,3] + 72.792;
   1:L PR[91] R[100]mm/sec CNT100;
   1:  PR[91,1] = PR[90,1] + -14.423;
   1:  PR[91,2] = PR[90,2] + 22.242;
   1:  PR[91,3] = PR[90,3] + 72.808;
   1:L PR[91] R[100]mm/sec CNT100;
   1:  PR[91,1] = PR[90,1] + -17.559;
   1:  PR[91,2] = PR[90,2] + 22.671;
   1:  PR[91,3] = PR[90,3] + 72.825;
   1:L PR[91] R[100]mm/sec CNT100;
   1:  PR[91,1] = PR[90,1] + -24.454;
   1:  PR[91,2] = PR[90,2] + 23.425;
   1:  PR[91,3] = PR[90,3] + 72.836;
   1:L PR[91] R[100]mm/sec CNT100;
   1:  PR[91,1] = PR[90,1] + -24.988;
   1:  PR[91,2] = PR[90,2] + 23.474;
   1:  PR[91,3] = PR[90,3] + 72.862;
   1:L PR[91] R[100]mm/sec CNT100;
   1:  PR[91,1] = PR[90,1] + -27.189;
   1:  PR[91,2] = PR[90,2] + 23.557;
   1:  PR[91,3] = PR[90,3] + 72.864;
   1:L PR[91] R[100]mm/sec CNT100;
   1:  PR[91,1] = PR[90,1] + -36.501;
   1:  PR[91,2] = PR[90,2] + 23.825;
   1:  PR[91,3] = PR[90,3] + 72.872;
   1:L PR[91] R[100]mm/sec CNT100;
   1:  PR[91,1] = PR[90,1] + -43.578;
   1:  PR[91,2] = PR[90,2] + 23.358;
   1:  PR[91,3] = PR[90,3] + 72.907;
   1:L PR[91] R[100]mm/sec CNT100;
   1:  PR[91,1] = PR[90,1] + -49.857;
   1:  PR[91,2] = PR[90,2] + 22.298;
   1:  PR[91,3] = PR[90,3] + 72.933;
   1:L PR[91] R[100]mm/sec CNT100;
   1:  PR[91,1] = PR[90,1] + -51.705;
   1:  PR[91,2] = PR[90,2] + 21.919;
   1:  PR[91,3] = PR[90,3] + 72.957;
   1:L PR[91] R[100]mm/sec CNT100;
   1:  PR[91,1] = PR[90,1] + -54.751;
   1:  PR[91,2] = PR[90,2] + 20.923;
   1:  PR[91,3] = PR[90,3] + 72.964;
   1:L PR[91] R[100]mm/sec CNT100;
   1:  PR[91,1] = PR[90,1] + -59.398;
   1:  PR[91,2] = PR[90,2] + 19.232;
   1:  PR[91,3] = PR[90,3] + 72.976;
   1:L PR[91] R[100]mm/sec CNT100;
   1:  PR[91,1] = PR[90,1] + -59.600;
   1:  PR[91,2] = PR[90,2] + 19.121;
   1:  PR[91,3] = PR[90,3] + 72.994;
   1:L PR[91] R[100]mm/sec CNT100;
   1:  PR[91] = PR[90];
   1:  PR[91,1] = PR[90,1] + -60.911;
   1:  PR[91,2] = PR[90,2] + 17.831;
   1:  PR[91,3] = PR[90,3] + 74.295;
   1:L PR[91] R[100]mm/sec CNT100;
   1:  PR[91,1] = PR[90,1] + -63.605;
   1:  PR[91,2] = PR[90,2] + 16.188;
   1:  PR[91,3] = PR[90,3] + 73.004;
   1:L PR[91] R[100]mm/sec CNT100;
   1:  PR[91,1] = PR[90,1] + -67.777;
   1:  PR[91,2] = PR[90,2] + 12.385;
   1:  PR[91,3] = PR[90,3] + 73.016;
   1:L PR[91] R[100]mm/sec CNT100;
   1:  PR[91,1] = PR[90,1] + -70.758;
   1:  PR[91,2] = PR[90,2] + 8.199;
   1:  PR[91,3] = PR[90,3] + 73.037;
   1:L PR[91] R[100]mm/sec CNT100;
   1:  PR[91,1] = PR[90,1] + -72.537;
   1:  PR[91,2] = PR[90,2] + 3.785;
   1:  PR[91,3] = PR[90,3] + 73.056;
   1:L PR[91] R[100]mm/sec CNT100;
   1:  PR[91,1] = PR[90,1] + -73.033;
   1:  PR[91,2] = PR[90,2] + -0.004;
   1:  PR[91,3] = PR[90,3] + 73.074;
   1:L PR[91] R[100]mm/sec CNT100;
   1:  PR[91,1] = PR[90,1] + -73.156;
   1:  PR[91,2] = PR[90,2] + -0.698;
   1:  PR[91,3] = PR[90,3] + 73.089;
   1:L PR[91] R[100]mm/sec CNT100;
   1:  PR[91,1] = PR[90,1] + -72.777;
   1:  PR[91,2] = PR[90,2] + -2.521;
   1:  PR[91,3] = PR[90,3] + 73.091;
   1:L PR[91] R[100]mm/sec CNT100;
   1:  PR[91,1] = PR[90,1] + -72.405;
   1:  PR[91,2] = PR[90,2] + -5.414;
   1:  PR[91,3] = PR[90,3] + 73.098;
   1:L PR[91] R[100]mm/sec CNT100;
   1:  PR[91,1] = PR[90,1] + -71.119;
   1:  PR[91,2] = PR[90,2] + -8.619;
   1:  PR[91,3] = PR[90,3] + 73.109;
   1:L PR[91] R[100]mm/sec CNT100;
   1:  PR[91,1] = PR[90,1] + -70.578;
   1:  PR[91,2] = PR[90,2] + -9.947;
   1:  PR[91,3] = PR[90,3] + 73.122;
   1:L PR[91] R[100]mm/sec CNT100;
   1:  PR[91,1] = PR[90,1] + -67.553;
   1:  PR[91,2] = PR[90,2] + -14.191;
   1:  PR[91,3] = PR[90,3] + 73.127;
   1:L PR[91] R[100]mm/sec CNT100;
   1:  PR[91,1] = PR[90,1] + -65.728;
   1:  PR[91,2] = PR[90,2] + -15.844;
   1:  PR[91,3] = PR[90,3] + 73.147;
   1:L PR[91] R[100]mm/sec CNT100;
   1:  PR[91,1] = PR[90,1] + -63.351;
   1:  PR[91,2] = PR[90,2] + -17.826;
   1:  PR[91,3] = PR[90,3] + 73.156;
   1:L PR[91] R[100]mm/sec CNT100;
   1:  PR[91,1] = PR[90,1] + -62.402;
   1:  PR[91,2] = PR[90,2] + -18.408;
   1:  PR[91,3] = PR[90,3] + 73.168;
   1:L PR[91] R[100]mm/sec CNT100;
   1:  PR[91,1] = PR[90,1] + -58.268;
   1:  PR[91,2] = PR[90,2] + -20.710;
   1:  PR[91,3] = PR[90,3] + 73.172;
   1:L PR[91] R[100]mm/sec CNT100;
   1:  PR[91,1] = PR[90,1] + -54.059;
   1:  PR[91,2] = PR[90,2] + -22.425;
   1:  PR[91,3] = PR[90,3] + 73.190;
   1:L PR[91] R[100]mm/sec CNT100;
   1:  PR[91,1] = PR[90,1] + -52.795;
   1:  PR[91,2] = PR[90,2] + -22.875;
   1:  PR[91,3] = PR[90,3] + 73.207;
   1:L PR[91] R[100]mm/sec CNT100;
   1:  PR[91,1] = PR[90,1] + -50.854;
   1:  PR[91,2] = PR[90,2] + -23.345;
   1:  PR[91,3] = PR[90,3] + 73.212;
   1:L PR[91] R[100]mm/sec CNT100;
   1:  PR[91,1] = PR[90,1] + -47.243;
   1:  PR[91,2] = PR[90,2] + -24.177;
   1:  PR[91,3] = PR[90,3] + 73.219;
   1:L PR[91] R[100]mm/sec CNT100;
   1:  PR[91,1] = PR[90,1] + -44.582;
   1:  PR[91,2] = PR[90,2] + -24.700;
   1:  PR[91,3] = PR[90,3] + 73.233;
   1:L PR[91] R[100]mm/sec CNT100;
   1:  PR[91,1] = PR[90,1] + -41.757;
   1:  PR[91,2] = PR[90,2] + -24.997;
   1:  PR[91,3] = PR[90,3] + 73.243;
   1:L PR[91] R[100]mm/sec CNT100;
   1:  PR[91,1] = PR[90,1] + -38.433;
   1:  PR[91,2] = PR[90,2] + -25.218;
   1:  PR[91,3] = PR[90,3] + 73.254;
   1:L PR[91] R[100]mm/sec CNT100;
   1:  PR[91,1] = PR[90,1] + -35.329;
   1:  PR[91,2] = PR[90,2] + -25.466;
   1:  PR[91,3] = PR[90,3] + 73.266;
   1:L PR[91] R[100]mm/sec CNT100;
   1:  PR[91,1] = PR[90,1] + -32.441;
   1:  PR[91,2] = PR[90,2] + -25.552;
   1:  PR[91,3] = PR[90,3] + 73.278;
   1:L PR[91] R[100]mm/sec CNT100;
   1:  PR[91,1] = PR[90,1] + -29.752;
   1:  PR[91,2] = PR[90,2] + -25.470;
   1:  PR[91,3] = PR[90,3] + 73.289;
   1:L PR[91] R[100]mm/sec CNT100;
   1:  PR[91,1] = PR[90,1] + -22.134;
   1:  PR[91,2] = PR[90,2] + -25.177;
   1:  PR[91,3] = PR[90,3] + 73.299;
   1:L PR[91] R[100]mm/sec CNT100;
   1:  PR[91,1] = PR[90,1] + -15.897;
   1:  PR[91,2] = PR[90,2] + -24.469;
   1:  PR[91,3] = PR[90,3] + 73.328;
   1:L PR[91] R[100]mm/sec CNT100;
   1:  PR[91,1] = PR[90,1] + -15.267;
   1:  PR[91,2] = PR[90,2] + -24.448;
   1:  PR[91,3] = PR[90,3] + 73.351;
   1:L PR[91] R[100]mm/sec CNT100;
   1:  PR[91,1] = PR[90,1] + -12.819;
   1:  PR[91,2] = PR[90,2] + -24.115;
   1:  PR[91,3] = PR[90,3] + 73.354;
   1:L PR[91] R[100]mm/sec CNT100;
   1:  PR[91,1] = PR[90,1] + -9.318;
   1:  PR[91,2] = PR[90,2] + -24.934;
   1:  PR[91,3] = PR[90,3] + 73.363;
   1:L PR[91] R[100]mm/sec CNT100;
   1:  PR[91,1] = PR[90,1] + -4.080;
   1:  PR[91,2] = PR[90,2] + -25.439;
   1:  PR[91,3] = PR[90,3] + 73.376;
   1:L PR[91] R[100]mm/sec CNT100;
   1:  PR[91,1] = PR[90,1] + -3.098;
   1:  PR[91,2] = PR[90,2] + -25.518;
   1:  PR[91,3] = PR[90,3] + 73.396;
   1:L PR[91] R[100]mm/sec CNT100;
   1:  PR[91,1] = PR[90,1] + -0.263;
   1:  PR[91,2] = PR[90,2] + -25.271;
   1:  PR[91,3] = PR[90,3] + 73.400;
   1:L PR[91] R[100]mm/sec CNT100;
   1:  PR[91,1] = PR[90,1] + 3.076;
   1:  PR[91,2] = PR[90,2] + -25.040;
   1:  PR[91,3] = PR[90,3] + 73.410;
   1:L PR[91] R[100]mm/sec CNT100;
   1:  PR[91,1] = PR[90,1] + 3.877;
   1:  PR[91,2] = PR[90,2] + -24.945;
   1:  PR[91,3] = PR[90,3] + 73.423;
   1:L PR[91] R[100]mm/sec CNT100;
   1:  PR[91,1] = PR[90,1] + 3.950;
   1:  PR[91,2] = PR[90,2] + -24.930;
   1:  PR[91,3] = PR[90,3] + 73.426;
   1:L PR[91] R[100]mm/sec CNT100;
   1:  PR[91,1] = PR[90,1] + 8.541;
   1:  PR[91,2] = PR[90,2] + -23.752;
   1:L PR[91] R[100]mm/sec CNT100;
   1:  PR[91,1] = PR[90,1] + 10.937;
   1:  PR[91,2] = PR[90,2] + -24.852;
   1:  PR[91,3] = PR[90,3] + 73.444;
   1:L PR[91] R[100]mm/sec CNT100;
   1:  PR[91,1] = PR[90,1] + 12.957;
   1:  PR[91,2] = PR[90,2] + -25.403;
   1:  PR[91,3] = PR[90,3] + 73.454;
   1:L PR[91] R[100]mm/sec CNT100;
   1:  PR[91,1] = PR[90,1] + 16.946;
   1:  PR[91,2] = PR[90,2] + -26.263;
   1:  PR[91,3] = PR[90,3] + 73.462;
   1:L PR[91] R[100]mm/sec CNT100;
   1:  PR[91,1] = PR[90,1] + 19.390;
   1:  PR[91,2] = PR[90,2] + -26.362;
   1:  PR[91,3] = PR[90,3] + 73.477;
   1:L PR[91] R[100]mm/sec CNT100;
   1:  PR[91,1] = PR[90,1] + 23.020;
   1:  PR[91,2] = PR[90,2] + -26.246;
   1:  PR[91,3] = PR[90,3] + 73.486;
   1:L PR[91] R[100]mm/sec CNT100;
   1:  PR[91,1] = PR[90,1] + 26.166;
   1:  PR[91,2] = PR[90,2] + -25.768;
   1:  PR[91,3] = PR[90,3] + 73.500;
   1:L PR[91] R[100]mm/sec CNT100;
   1:  PR[91,1] = PR[90,1] + 30.789;
   1:  PR[91,2] = PR[90,2] + -26.975;
   1:  PR[91,3] = PR[90,3] + 73.512;
   1:L PR[91] R[100]mm/sec CNT100;
   1:  PR[91,1] = PR[90,1] + 31.389;
   1:  PR[91,2] = PR[90,2] + -27.119;
   1:  PR[91,3] = PR[90,3] + 73.530;
   1:L PR[91] R[100]mm/sec CNT100;
   1:  PR[91,1] = PR[90,1] + 31.607;
   1:  PR[91,2] = PR[90,2] + -27.149;
   1:  PR[91,3] = PR[90,3] + 73.532;
   1:L PR[91] R[100]mm/sec CNT100;
   1:  PR[91,1] = PR[90,1] + 36.451;
   1:  PR[91,2] = PR[90,2] + -27.543;
   1:  PR[91,3] = PR[90,3] + 73.533;
   1:L PR[91] R[100]mm/sec CNT100;
   1:  PR[91,1] = PR[90,1] + 39.115;
   1:  PR[91,2] = PR[90,2] + -27.498;
   1:  PR[91,3] = PR[90,3] + 73.551;
   1:L PR[91] R[100]mm/sec CNT100;
   1:  PR[91,1] = PR[90,1] + 41.086;
   1:  PR[91,2] = PR[90,2] + -27.346;
   1:  PR[91,3] = PR[90,3] + 73.561;
   1:L PR[91] R[100]mm/sec CNT100;
   1:  PR[91,1] = PR[90,1] + 44.077;
   1:  PR[91,2] = PR[90,2] + -26.831;
   1:  PR[91,3] = PR[90,3] + 73.569;
   1:L PR[91] R[100]mm/sec CNT100;
   1:  PR[91,1] = PR[90,1] + 45.841;
   1:  PR[91,2] = PR[90,2] + -26.594;
   1:  PR[91,3] = PR[90,3] + 73.580;
   1:L PR[91] R[100]mm/sec CNT100;
   1:  PR[91,1] = PR[90,1] + 47.415;
   1:  PR[91,2] = PR[90,2] + -26.203;
   1:  PR[91,3] = PR[90,3] + 73.587;
   1:L PR[91] R[100]mm/sec CNT100;
   1:  PR[91,1] = PR[90,1] + 50.701;
   1:  PR[91,2] = PR[90,2] + -25.316;
   1:  PR[91,3] = PR[90,3] + 73.593;
   1:L PR[91] R[100]mm/sec CNT100;
   1:  PR[91,1] = PR[90,1] + 53.247;
   1:  PR[91,2] = PR[90,2] + -24.327;
   1:  PR[91,3] = PR[90,3] + 73.605;
   1:L PR[91] R[100]mm/sec CNT100;
   1:  PR[91,1] = PR[90,1] + 55.044;
   1:  PR[91,2] = PR[90,2] + -23.740;
   1:  PR[91,3] = PR[90,3] + 73.616;
   1:L PR[91] R[100]mm/sec CNT100;
   1:  PR[91,1] = PR[90,1] + 59.326;
   1:  PR[91,2] = PR[90,2] + -21.797;
   1:  PR[91,3] = PR[90,3] + 73.623;
   1:L PR[91] R[100]mm/sec CNT100;
   1:  PR[91,1] = PR[90,1] + 63.257;
   1:  PR[91,2] = PR[90,2] + -19.293;
   1:  PR[91,3] = PR[90,3] + 73.640;
   1:L PR[91] R[100]mm/sec CNT100;
   1:  PR[91,1] = PR[90,1] + 64.999;
   1:  PR[91,2] = PR[90,2] + -17.857;
   1:  PR[91,3] = PR[90,3] + 73.658;
   1:L PR[91] R[100]mm/sec CNT100;
   1:  PR[91,1] = PR[90,1] + 67.258;
   1:  PR[91,2] = PR[90,2] + -15.869;
   1:  PR[91,3] = PR[90,3] + 73.666;
   1:L PR[91] R[100]mm/sec CNT100;
   1:  PR[91,1] = PR[90,1] + 69.969;
   1:  PR[91,2] = PR[90,2] + -12.422;
   1:  PR[91,3] = PR[90,3] + 73.678;
   1:L PR[91] R[100]mm/sec CNT100;
   1:  PR[91,1] = PR[90,1] + 70.849;
   1:  PR[91,2] = PR[90,2] + -11.330;
   1:  PR[91,3] = PR[90,3] + 73.694;
   1:L PR[91] R[100]mm/sec CNT100;
   1:  PR[91,1] = PR[90,1] + 71.207;
   1:  PR[91,2] = PR[90,2] + -10.686;
   1:  PR[91,3] = PR[90,3] + 73.699;
   1:L PR[91] R[100]mm/sec CNT100;
   1:  PR[91,1] = PR[90,1] + 73.223;
   1:  PR[91,2] = PR[90,2] + -6.082;
   1:  PR[91,3] = PR[90,3] + 73.702;
   1:L PR[91] R[100]mm/sec CNT100;
   1:  PR[91,1] = PR[90,1] + 73.252;
   1:  PR[91,2] = PR[90,2] + -5.992;
   1:  PR[91,3] = PR[90,3] + 73.721;
   1:L PR[91] R[100]mm/sec CNT100;
   1:  PR[91,1] = PR[90,1] + 74.000;
   1:  PR[91,2] = PR[90,2] + -0.732;
   1:L PR[91] R[100]mm/sec CNT100;
   1:  PR[91,1] = PR[90,1] + 73.258;
   1:  PR[91,2] = PR[90,2] + 4.411;
   1:  PR[91,3] = PR[90,3] + 73.741;
   1:L PR[91] R[100]mm/sec CNT100;
   1:  PR[91,1] = PR[90,1] + 73.242;
   1:  PR[91,2] = PR[90,2] + 4.566;
   1:  PR[91,3] = PR[90,3] + 73.761;
   1:L PR[91] R[100]mm/sec CNT100;
   1:  PR[91,1] = PR[90,1] + 73.224;
   1:  PR[91,2] = PR[90,2] + 4.620;
   1:L PR[91] R[100]mm/sec CNT100;
   1:  PR[91,1] = PR[90,1] + 71.210;
   1:  PR[91,2] = PR[90,2] + 9.223;
   1:  PR[91,3] = PR[90,3] + 73.762;
   1:L PR[91] R[100]mm/sec CNT100;
   1:  PR[91,1] = PR[90,1] + 70.845;
   1:  PR[91,2] = PR[90,2] + 9.879;
   1:  PR[91,3] = PR[90,3] + 73.780;
   1:L PR[91] R[100]mm/sec CNT100;
   1:  PR[91,1] = PR[90,1] + 68.354;
   1:  PR[91,2] = PR[90,2] + 13.068;
   1:  PR[91,3] = PR[90,3] + 73.783;
   1:L PR[91] R[100]mm/sec CNT100;
   1:  PR[91,1] = PR[90,1] + 67.275;
   1:  PR[91,2] = PR[90,2] + 14.395;
   1:  PR[91,3] = PR[90,3] + 73.798;
   1:L PR[91] R[100]mm/sec CNT100;
   1:  PR[91,1] = PR[90,1] + 65.003;
   1:  PR[91,2] = PR[90,2] + 16.394;
   1:  PR[91,3] = PR[90,3] + 73.805;
   1:L PR[91] R[100]mm/sec CNT100;
   1:  PR[91,1] = PR[90,1] + 63.260;
   1:  PR[91,2] = PR[90,2] + 17.832;
   1:  PR[91,3] = PR[90,3] + 73.816;
   1:L PR[91] R[100]mm/sec CNT100;
   1:  PR[91,1] = PR[90,1] + 59.326;
   1:  PR[91,2] = PR[90,2] + 20.338;
   1:  PR[91,3] = PR[90,3] + 73.825;
   1:L PR[91] R[100]mm/sec CNT100;
   1:  PR[91,1] = PR[90,1] + 55.044;
   1:  PR[91,2] = PR[90,2] + 22.281;
   1:  PR[91,3] = PR[90,3] + 73.842;
   1:L PR[91] R[100]mm/sec CNT100;
   1:  PR[91,1] = PR[90,1] + 53.247;
   1:  PR[91,2] = PR[90,2] + 22.869;
   1:  PR[91,3] = PR[90,3] + 73.860;
   1:L PR[91] R[100]mm/sec CNT100;
   1:  PR[91,1] = PR[90,1] + 50.701;
   1:  PR[91,2] = PR[90,2] + 23.857;
   1:  PR[91,3] = PR[90,3] + 73.867;
   1:L PR[91] R[100]mm/sec CNT100;
   1:  PR[91,1] = PR[90,1] + 47.416;
   1:  PR[91,2] = PR[90,2] + 24.744;
   1:  PR[91,3] = PR[90,3] + 73.877;
   1:L PR[91] R[100]mm/sec CNT100;
   1:  PR[91,1] = PR[90,1] + 45.841;
   1:  PR[91,2] = PR[90,2] + 25.135;
   1:  PR[91,3] = PR[90,3] + 73.890;
   1:L PR[91] R[100]mm/sec CNT100;
   1:  PR[91,1] = PR[90,1] + 44.077;
   1:  PR[91,2] = PR[90,2] + 25.372;
   1:  PR[91,3] = PR[90,3] + 73.896;
   1:L PR[91] R[100]mm/sec CNT100;
   1:  PR[91,1] = PR[90,1] + 41.086;
   1:  PR[91,2] = PR[90,2] + 25.887;
   1:  PR[91,3] = PR[90,3] + 73.903;
   1:L PR[91] R[100]mm/sec CNT100;
   1:  PR[91,1] = PR[90,1] + 39.115;
   1:  PR[91,2] = PR[90,2] + 26.039;
   1:  PR[91,3] = PR[90,3] + 73.914;
   1:L PR[91] R[100]mm/sec CNT100;
   1:  PR[91,1] = PR[90,1] + 36.451;
   1:  PR[91,2] = PR[90,2] + 26.084;
   1:  PR[91,3] = PR[90,3] + 73.921;
   1:L PR[91] R[100]mm/sec CNT100;
   1:  PR[91,1] = PR[90,1] + 31.607;
   1:  PR[91,2] = PR[90,2] + 25.690;
   1:  PR[91,3] = PR[90,3] + 73.931;
   1:L PR[91] R[100]mm/sec CNT100;
   1:  PR[91,1] = PR[90,1] + 31.390;
   1:  PR[91,2] = PR[90,2] + 25.660;
   1:  PR[91,3] = PR[90,3] + 73.950;
   1:L PR[91] R[100]mm/sec CNT100;
   1:  PR[91,1] = PR[90,1] + 30.789;
   1:  PR[91,2] = PR[90,2] + 25.516;
   1:L PR[91] R[100]mm/sec CNT100;
   1:  PR[91,1] = PR[90,1] + 26.166;
   1:  PR[91,2] = PR[90,2] + 24.310;
   1:  PR[91,3] = PR[90,3] + 73.953;
   1:L PR[91] R[100]mm/sec CNT100;
   1:  PR[91,1] = PR[90,1] + 23.020;
   1:  PR[91,2] = PR[90,2] + 24.787;
   1:  PR[91,3] = PR[90,3] + 73.971;
   1:L PR[91] R[100]mm/sec CNT100;
   1:  PR[91,1] = PR[90,1] + 19.389;
   1:  PR[91,2] = PR[90,2] + 24.904;
   1:  PR[91,3] = PR[90,3] + 73.983;
   1:L PR[91] R[100]mm/sec CNT100;
   1:  PR[91,1] = PR[90,1] + 16.945;
   1:  PR[91,2] = PR[90,2] + 24.804;
   1:  PR[91,3] = PR[90,3] + 73.996;
   1:L PR[91] R[100]mm/sec CNT100;
   1:  PR[91,1] = PR[90,1] + 12.957;
   1:  PR[91,2] = PR[90,2] + 23.944;
   1:  PR[91,3] = PR[90,3] + 74.005;
   1:L PR[91] R[100]mm/sec CNT100;
   1:  PR[91,1] = PR[90,1] + 10.936;
   1:  PR[91,2] = PR[90,2] + 23.393;
   1:  PR[91,3] = PR[90,3] + 74.021;
   1:L PR[91] R[100]mm/sec CNT100;
   1:  PR[91,1] = PR[90,1] + 8.540;
   1:  PR[91,2] = PR[90,2] + 22.294;
   1:  PR[91,3] = PR[90,3] + 74.029;
   1:L PR[91] R[100]mm/sec CNT100;
   1:  PR[91,1] = PR[90,1] + 3.990;
   1:  PR[91,2] = PR[90,2] + 23.465;
   1:  PR[91,3] = PR[90,3] + 74.038;
   1:L PR[91] R[100]mm/sec CNT100;
   1:  PR[91,1] = PR[90,1] + 3.918;
   1:  PR[91,2] = PR[90,2] + 23.480;
   1:  PR[91,3] = PR[90,3] + 74.056;
   1:L PR[91] R[100]mm/sec CNT100;
   1:  PR[91,1] = PR[90,1] + 3.110;
   1:  PR[91,2] = PR[90,2] + 23.575;
   1:L PR[91] R[100]mm/sec CNT100;
   1:  PR[91,1] = PR[90,1] + -0.265;
   1:  PR[91,2] = PR[90,2] + 23.811;
   1:  PR[91,3] = PR[90,3] + 74.059;
   1:L PR[91] R[100]mm/sec CNT100;
   1:  PR[91,1] = PR[90,1] + -3.075;
   1:  PR[91,2] = PR[90,2] + 24.060;
   1:  PR[91,3] = PR[90,3] + 74.072;
   1:L PR[91] R[100]mm/sec CNT100;
   1:  PR[91,1] = PR[90,1] + -4.049;
   1:  PR[91,2] = PR[90,2] + 23.981;
   1:  PR[91,3] = PR[90,3] + 74.083;
   1:L PR[91] R[100]mm/sec CNT100;
   1:  PR[91,1] = PR[90,1] + -9.316;
   1:  PR[91,2] = PR[90,2] + 23.475;
   1:  PR[91,3] = PR[90,3] + 74.086;
   1:L PR[91] R[100]mm/sec CNT100;
   1:  PR[91,1] = PR[90,1] + -12.817;
   1:  PR[91,2] = PR[90,2] + 22.655;
   1:  PR[91,3] = PR[90,3] + 74.106;
   1:L PR[91] R[100]mm/sec CNT100;
   1:  PR[91,1] = PR[90,1] + -15.342;
   1:  PR[91,2] = PR[90,2] + 22.999;
   1:  PR[91,3] = PR[90,3] + 74.120;
   1:L PR[91] R[100]mm/sec CNT100;
   1:  PR[91,1] = PR[90,1] + -20.795;
   1:  PR[91,2] = PR[90,2] + 23.595;
   1:  PR[91,3] = PR[90,3] + 74.129;
   1:L PR[91] R[100]mm/sec CNT100;
   1:  PR[91,1] = PR[90,1] + -22.236;
   1:  PR[91,2] = PR[90,2] + 23.727;
   1:  PR[91,3] = PR[90,3] + 74.150;
   1:L PR[91] R[100]mm/sec CNT100;
   1:  PR[91,1] = PR[90,1] + -27.838;
   1:  PR[91,2] = PR[90,2] + 23.938;
   1:  PR[91,3] = PR[90,3] + 74.155;
   1:L PR[91] R[100]mm/sec CNT100;
   1:  PR[91,1] = PR[90,1] + -33.003;
   1:  PR[91,2] = PR[90,2] + 24.087;
   1:  PR[91,3] = PR[90,3] + 74.176;
   1:L PR[91] R[100]mm/sec CNT100;
   1:  PR[91,1] = PR[90,1] + -35.299;
   1:  PR[91,2] = PR[90,2] + 24.022;
   1:  PR[91,3] = PR[90,3] + 74.196;
   1:L PR[91] R[100]mm/sec CNT100;
   1:  PR[91,1] = PR[90,1] + -37.275;
   1:  PR[91,2] = PR[90,2] + 23.854;
   1:  PR[91,3] = PR[90,3] + 74.204;
   1:L PR[91] R[100]mm/sec CNT100;
   1:  PR[91,1] = PR[90,1] + -42.440;
   1:  PR[91,2] = PR[90,2] + 23.513;
   1:  PR[91,3] = PR[90,3] + 74.212;
   1:L PR[91] R[100]mm/sec CNT100;
   1:  PR[91,1] = PR[90,1] + -49.331;
   1:  PR[91,2] = PR[90,2] + 22.340;
   1:  PR[91,3] = PR[90,3] + 74.231;
   1:L PR[91] R[100]mm/sec CNT100;
   1:  PR[91,1] = PR[90,1] + -50.017;
   1:  PR[91,2] = PR[90,2] + 22.199;
   1:  PR[91,3] = PR[90,3] + 74.257;
   1:L PR[91] R[100]mm/sec CNT100;
   1:  PR[91,1] = PR[90,1] + -54.206;
   1:  PR[91,2] = PR[90,2] + 20.829;
   1:  PR[91,3] = PR[90,3] + 74.260;
   1:L PR[91] R[100]mm/sec CNT100;
   1:  PR[91,1] = PR[90,1] + -57.892;
   1:  PR[91,2] = PR[90,2] + 19.487;
   1:  PR[91,3] = PR[90,3] + 74.276;
   1:L PR[91] R[100]mm/sec CNT100;
   1:  PR[91,1] = PR[90,1] + -58.805;
   1:  PR[91,2] = PR[90,2] + 19.009;
   1:  PR[91,3] = PR[90,3] + 74.291;
   1:L PR[91] R[100]mm/sec CNT100;
   1:  PR[91] = PR[90];
   1:  PR[91,1] = PR[90,1] + -62.230;
   1:  PR[91,2] = PR[90,2] + 16.537;
   1:  PR[91,3] = PR[90,3] + 75.595;
   1:L PR[91] R[100]mm/sec CNT100;
   1:  PR[91,1] = PR[90,1] + -62.554;
   1:  PR[91,2] = PR[90,2] + 16.339;
   1:  PR[91,3] = PR[90,3] + 74.312;
   1:L PR[91] R[100]mm/sec CNT100;
   1:  PR[91,1] = PR[90,1] + -66.769;
   1:  PR[91,2] = PR[90,2] + 12.501;
   1:  PR[91,3] = PR[90,3] + 74.314;
   1:L PR[91] R[100]mm/sec CNT100;
   1:  PR[91,1] = PR[90,1] + -69.779;
   1:  PR[91,2] = PR[90,2] + 8.278;
   1:  PR[91,3] = PR[90,3] + 74.335;
   1:L PR[91] R[100]mm/sec CNT100;
   1:  PR[91,1] = PR[90,1] + -71.575;
   1:  PR[91,2] = PR[90,2] + 3.825;
   1:  PR[91,3] = PR[90,3] + 74.355;
   1:L PR[91] R[100]mm/sec CNT100;
   1:  PR[91,1] = PR[90,1] + -71.976;
   1:  PR[91,2] = PR[90,2] + 0.761;
   1:  PR[91,3] = PR[90,3] + 74.373;
   1:L PR[91] R[100]mm/sec CNT100;
   1:  PR[91,1] = PR[90,1] + -72.233;
   1:  PR[91,2] = PR[90,2] + -0.698;
   1:  PR[91,3] = PR[90,3] + 74.385;
   1:L PR[91] R[100]mm/sec CNT100;
   1:  PR[91,1] = PR[90,1] + -71.979;
   1:  PR[91,2] = PR[90,2] + -1.925;
   1:  PR[91,3] = PR[90,3] + 74.391;
   1:L PR[91] R[100]mm/sec CNT100;
   1:  PR[91,1] = PR[90,1] + -71.526;
   1:  PR[91,2] = PR[90,2] + -5.441;
   1:  PR[91,3] = PR[90,3] + 74.395;
   1:L PR[91] R[100]mm/sec CNT100;
   1:  PR[91,1] = PR[90,1] + -69.959;
   1:  PR[91,2] = PR[90,2] + -9.346;
   1:  PR[91,3] = PR[90,3] + 74.409;
   1:L PR[91] R[100]mm/sec CNT100;
   1:  PR[91,1] = PR[90,1] + -69.692;
   1:  PR[91,2] = PR[90,2] + -10.003;
   1:  PR[91,3] = PR[90,3] + 74.425;
   1:L PR[91] R[100]mm/sec CNT100;
   1:  PR[91,1] = PR[90,1] + -66.856;
   1:  PR[91,2] = PR[90,2] + -13.988;
   1:  PR[91,3] = PR[90,3] + 74.428;
   1:L PR[91] R[100]mm/sec CNT100;
   1:  PR[91,1] = PR[90,1] + -66.676;
   1:  PR[91,2] = PR[90,2] + -14.218;
   1:  PR[91,3] = PR[90,3] + 74.446;
   1:L PR[91] R[100]mm/sec CNT100;
   1:  PR[91,1] = PR[90,1] + -62.353;
   1:  PR[91,2] = PR[90,2] + -17.822;
   1:  PR[91,3] = PR[90,3] + 74.447;
   1:L PR[91] R[100]mm/sec CNT100;
   1:  PR[91,1] = PR[90,1] + -60.340;
   1:  PR[91,2] = PR[90,2] + -19.056;
   1:  PR[91,3] = PR[90,3] + 74.469;
   1:L PR[91] R[100]mm/sec CNT100;
   1:  PR[91,1] = PR[90,1] + -57.328;
   1:  PR[91,2] = PR[90,2] + -20.734;
   1:  PR[91,3] = PR[90,3] + 74.477;
   1:L PR[91] R[100]mm/sec CNT100;
   1:  PR[91,1] = PR[90,1] + -51.882;
   1:  PR[91,2] = PR[90,2] + -22.951;
   1:  PR[91,3] = PR[90,3] + 74.491;
   1:L PR[91] R[100]mm/sec CNT100;
   1:  PR[91,1] = PR[90,1] + -46.501;
   1:  PR[91,2] = PR[90,2] + -24.192;
   1:  PR[91,3] = PR[90,3] + 74.513;
   1:L PR[91] R[100]mm/sec CNT100;
   1:  PR[91,1] = PR[90,1] + -42.429;
   1:  PR[91,2] = PR[90,2] + -24.992;
   1:  PR[91,3] = PR[90,3] + 74.534;
   1:L PR[91] R[100]mm/sec CNT100;
   1:  PR[91,1] = PR[90,1] + -41.016;
   1:  PR[91,2] = PR[90,2] + -25.140;
   1:  PR[91,3] = PR[90,3] + 74.550;
   1:L PR[91] R[100]mm/sec CNT100;
   1:  PR[91,1] = PR[90,1] + -39.295;
   1:  PR[91,2] = PR[90,2] + -25.255;
   1:  PR[91,3] = PR[90,3] + 74.555;
   1:L PR[91] R[100]mm/sec CNT100;
   1:  PR[91,1] = PR[90,1] + -34.170;
   1:  PR[91,2] = PR[90,2] + -25.663;
   1:  PR[91,3] = PR[90,3] + 74.561;
   1:L PR[91] R[100]mm/sec CNT100;
   1:  PR[91,1] = PR[90,1] + -29.360;
   1:  PR[91,2] = PR[90,2] + -25.808;
   1:  PR[91,3] = PR[90,3] + 74.581;
   1:L PR[91] R[100]mm/sec CNT100;
   1:  PR[91,1] = PR[90,1] + -19.571;
   1:  PR[91,2] = PR[90,2] + -25.445;
   1:  PR[91,3] = PR[90,3] + 74.599;
   1:L PR[91] R[100]mm/sec CNT100;
   1:  PR[91,1] = PR[90,1] + -19.341;
   1:  PR[91,2] = PR[90,2] + -25.428;
   1:  PR[91,3] = PR[90,3] + 74.636;
   1:L PR[91] R[100]mm/sec CNT100;
   1:  PR[91,1] = PR[90,1] + -13.828;
   1:  PR[91,2] = PR[90,2] + -24.802;
   1:  PR[91,3] = PR[90,3] + 74.637;
   1:L PR[91] R[100]mm/sec CNT100;
   1:  PR[91,1] = PR[90,1] + -13.051;
   1:  PR[91,2] = PR[90,2] + -24.776;
   1:  PR[91,3] = PR[90,3] + 74.658;
   1:L PR[91] R[100]mm/sec CNT100;
   1:  PR[91,1] = PR[90,1] + -11.210;
   1:  PR[91,2] = PR[90,2] + -24.526;
   1:  PR[91,3] = PR[90,3] + 74.661;
   1:L PR[91] R[100]mm/sec CNT100;
   1:  PR[91,1] = PR[90,1] + -8.621;
   1:  PR[91,2] = PR[90,2] + -25.132;
   1:  PR[91,3] = PR[90,3] + 74.668;
   1:L PR[91] R[100]mm/sec CNT100;
   1:  PR[91,1] = PR[90,1] + -2.308;
   1:  PR[91,2] = PR[90,2] + -25.739;
   1:  PR[91,3] = PR[90,3] + 74.678;
   1:L PR[91] R[100]mm/sec CNT100;
   1:  PR[91,1] = PR[90,1] + 3.588;
   1:  PR[91,2] = PR[90,2] + -25.327;
   1:  PR[91,3] = PR[90,3] + 74.702;
   1:L PR[91] R[100]mm/sec CNT100;
   1:  PR[91,1] = PR[90,1] + 5.072;
   1:  PR[91,2] = PR[90,2] + -25.151;
   1:  PR[91,3] = PR[90,3] + 74.725;
   1:L PR[91] R[100]mm/sec CNT100;
   1:  PR[91,1] = PR[90,1] + 5.294;
   1:  PR[91,2] = PR[90,2] + -25.106;
   1:  PR[91,3] = PR[90,3] + 74.730;
   1:L PR[91] R[100]mm/sec CNT100;
   1:  PR[91,1] = PR[90,1] + 8.887;
   1:  PR[91,2] = PR[90,2] + -24.184;
   1:  PR[91,3] = PR[90,3] + 74.731;
   1:L PR[91] R[100]mm/sec CNT100;
   1:  PR[91,1] = PR[90,1] + 10.803;
   1:  PR[91,2] = PR[90,2] + -25.064;
   1:  PR[91,3] = PR[90,3] + 74.745;
   1:L PR[91] R[100]mm/sec CNT100;
   1:  PR[91,1] = PR[90,1] + 12.260;
   1:  PR[91,2] = PR[90,2] + -25.461;
   1:  PR[91,3] = PR[90,3] + 74.753;
   1:L PR[91] R[100]mm/sec CNT100;
   1:  PR[91,1] = PR[90,1] + 16.908;
   1:  PR[91,2] = PR[90,2] + -26.464;
   1:  PR[91,3] = PR[90,3] + 74.759;
   1:L PR[91] R[100]mm/sec CNT100;
   1:  PR[91,1] = PR[90,1] + 18.784;
   1:  PR[91,2] = PR[90,2] + -26.540;
   1:  PR[91,3] = PR[90,3] + 74.777;
   1:L PR[91] R[100]mm/sec CNT100;
   1:  PR[91,1] = PR[90,1] + 23.071;
   1:  PR[91,2] = PR[90,2] + -26.402;
   1:  PR[91,3] = PR[90,3] + 74.784;
   1:L PR[91] R[100]mm/sec CNT100;
   1:  PR[91,1] = PR[90,1] + 25.698;
   1:  PR[91,2] = PR[90,2] + -26.004;
   1:  PR[91,3] = PR[90,3] + 74.800;
   1:L PR[91] R[100]mm/sec CNT100;
   1:  PR[91,1] = PR[90,1] + 30.362;
   1:  PR[91,2] = PR[90,2] + -27.222;
   1:  PR[91,3] = PR[90,3] + 74.811;
   1:L PR[91] R[100]mm/sec CNT100;
   1:  PR[91,1] = PR[90,1] + 30.917;
   1:  PR[91,2] = PR[90,2] + -27.349;
   1:  PR[91,3] = PR[90,3] + 74.829;
   1:L PR[91] R[100]mm/sec CNT100;
   1:  PR[91,1] = PR[90,1] + 36.092;
   1:  PR[91,2] = PR[90,2] + -27.767;
   1:  PR[91,3] = PR[90,3] + 74.831;
   1:L PR[91] R[100]mm/sec CNT100;
   1:  PR[91,1] = PR[90,1] + 37.562;
   1:  PR[91,2] = PR[90,2] + -27.742;
   1:  PR[91,3] = PR[90,3] + 74.851;
   1:L PR[91] R[100]mm/sec CNT100;
   1:  PR[91,1] = PR[90,1] + 40.843;
   1:  PR[91,2] = PR[90,2] + -27.489;
   1:  PR[91,3] = PR[90,3] + 74.856;
   1:L PR[91] R[100]mm/sec CNT100;
   1:  PR[91,1] = PR[90,1] + 44.859;
   1:  PR[91,2] = PR[90,2] + -26.798;
   1:  PR[91,3] = PR[90,3] + 74.869;
   1:L PR[91] R[100]mm/sec CNT100;
   1:  PR[91,1] = PR[90,1] + 45.035;
   1:  PR[91,2] = PR[90,2] + -26.755;
   1:  PR[91,3] = PR[90,3] + 74.884;
   1:L PR[91] R[100]mm/sec CNT100;
   1:  PR[91,1] = PR[90,1] + 45.439;
   1:  PR[91,2] = PR[90,2] + -26.620;
   1:  PR[91,3] = PR[90,3] + 74.885;
   1:L PR[91] R[100]mm/sec CNT100;
   1:  PR[91,1] = PR[90,1] + 50.066;
   1:  PR[91,2] = PR[90,2] + -25.370;
   1:  PR[91,3] = PR[90,3] + 74.886;
   1:L PR[91] R[100]mm/sec CNT100;
   1:  PR[91,1] = PR[90,1] + 54.222;
   1:  PR[91,2] = PR[90,2] + -23.752;
   1:  PR[91,3] = PR[90,3] + 74.905;
   1:L PR[91] R[100]mm/sec CNT100;
   1:  PR[91,1] = PR[90,1] + 58.483;
   1:  PR[91,2] = PR[90,2] + -21.746;
   1:  PR[91,3] = PR[90,3] + 74.922;
   1:L PR[91] R[100]mm/sec CNT100;
   1:  PR[91,1] = PR[90,1] + 60.714;
   1:  PR[91,2] = PR[90,2] + -20.361;
   1:  PR[91,3] = PR[90,3] + 74.939;
   1:L PR[91] R[100]mm/sec CNT100;
   1:  PR[91,1] = PR[90,1] + 62.441;
   1:  PR[91,2] = PR[90,2] + -19.259;
   1:  PR[91,3] = PR[90,3] + 74.949;
   1:L PR[91] R[100]mm/sec CNT100;
   1:  PR[91,1] = PR[90,1] + 63.212;
   1:  PR[91,2] = PR[90,2] + -18.624;
   1:  PR[91,3] = PR[90,3] + 74.957;
   1:L PR[91] R[100]mm/sec CNT100;
   1:  PR[91,1] = PR[90,1] + 66.249;
   1:  PR[91,2] = PR[90,2] + -15.952;
   1:  PR[91,3] = PR[90,3] + 74.961;
   1:L PR[91] R[100]mm/sec CNT100;
   1:  PR[91,1] = PR[90,1] + 68.196;
   1:  PR[91,2] = PR[90,2] + -13.476;
   1:  PR[91,3] = PR[90,3] + 74.976;
   1:L PR[91] R[100]mm/sec CNT100;
   1:  PR[91,1] = PR[90,1] + 69.716;
   1:  PR[91,2] = PR[90,2] + -11.590;
   1:  PR[91,3] = PR[90,3] + 74.988;
   1:L PR[91] R[100]mm/sec CNT100;
   1:  PR[91,1] = PR[90,1] + 70.392;
   1:  PR[91,2] = PR[90,2] + -10.373;
   1:  PR[91,3] = PR[90,3] + 74.997;
   1:L PR[91] R[100]mm/sec CNT100;
   1:  PR[91,1] = PR[90,1] + 72.069;
   1:  PR[91,2] = PR[90,2] + -6.543;
   1:  PR[91,3] = PR[90,3] + 75.003;
   1:L PR[91] R[100]mm/sec CNT100;
   1:  PR[91,1] = PR[90,1] + 72.303;
   1:  PR[91,2] = PR[90,2] + -5.816;
   1:  PR[91,3] = PR[90,3] + 75.018;
   1:L PR[91] R[100]mm/sec CNT100;
   1:  PR[91,1] = PR[90,1] + 72.956;
   1:  PR[91,2] = PR[90,2] + -1.250;
   1:  PR[91,3] = PR[90,3] + 75.021;
   1:L PR[91] R[100]mm/sec CNT100;
   1:  PR[91,1] = PR[90,1] + 73.007;
   1:  PR[91,2] = PR[90,2] + -0.768;
   1:  PR[91,3] = PR[90,3] + 75.039;
   1:L PR[91] R[100]mm/sec CNT100;
   1:  PR[91,1] = PR[90,1] + 72.370;
   1:  PR[91,2] = PR[90,2] + 3.645;
   1:  PR[91,3] = PR[90,3] + 75.041;
   1:L PR[91] R[100]mm/sec CNT100;
   1:  PR[91,1] = PR[90,1] + 72.292;
   1:  PR[91,2] = PR[90,2] + 4.391;
   1:  PR[91,3] = PR[90,3] + 75.058;
   1:L PR[91] R[100]mm/sec CNT100;
   1:  PR[91,1] = PR[90,1] + 72.070;
   1:  PR[91,2] = PR[90,2] + 5.082;
   1:  PR[91,3] = PR[90,3] + 75.060;
   1:L PR[91] R[100]mm/sec CNT100;
   1:  PR[91,1] = PR[90,1] + 70.395;
   1:  PR[91,2] = PR[90,2] + 8.910;
   1:  PR[91,3] = PR[90,3] + 75.063;
   1:L PR[91] R[100]mm/sec CNT100;
   1:  PR[91,1] = PR[90,1] + 69.711;
   1:  PR[91,2] = PR[90,2] + 10.140;
   1:  PR[91,3] = PR[90,3] + 75.079;
   1:L PR[91] R[100]mm/sec CNT100;
   1:  PR[91,1] = PR[90,1] + 67.727;
   1:  PR[91,2] = PR[90,2] + 12.678;
   1:  PR[91,3] = PR[90,3] + 75.084;
   1:L PR[91] R[100]mm/sec CNT100;
   1:  PR[91,1] = PR[90,1] + 66.264;
   1:  PR[91,2] = PR[90,2] + 14.479;
   1:  PR[91,3] = PR[90,3] + 75.097;
   1:L PR[91] R[100]mm/sec CNT100;
   1:  PR[91,1] = PR[90,1] + 63.214;
   1:  PR[91,2] = PR[90,2] + 17.163;
   1:  PR[91,3] = PR[90,3] + 75.105;
   1:L PR[91] R[100]mm/sec CNT100;
   1:  PR[91,1] = PR[90,1] + 62.442;
   1:  PR[91,2] = PR[90,2] + 17.799;
   1:  PR[91,3] = PR[90,3] + 75.121;
   1:L PR[91] R[100]mm/sec CNT100;
   1:  PR[91,1] = PR[90,1] + 60.714;
   1:  PR[91,2] = PR[90,2] + 18.902;
   1:  PR[91,3] = PR[90,3] + 75.125;
   1:L PR[91] R[100]mm/sec CNT100;
   1:  PR[91,1] = PR[90,1] + 58.483;
   1:  PR[91,2] = PR[90,2] + 20.287;
   1:  PR[91,3] = PR[90,3] + 75.132;
   1:L PR[91] R[100]mm/sec CNT100;
   1:  PR[91,1] = PR[90,1] + 54.222;
   1:  PR[91,2] = PR[90,2] + 22.293;
   1:  PR[91,3] = PR[90,3] + 75.142;
   1:L PR[91] R[100]mm/sec CNT100;
   1:  PR[91,1] = PR[90,1] + 50.066;
   1:  PR[91,2] = PR[90,2] + 23.911;
   1:  PR[91,3] = PR[90,3] + 75.160;
   1:L PR[91] R[100]mm/sec CNT100;
   1:  PR[91,1] = PR[90,1] + 45.439;
   1:  PR[91,2] = PR[90,2] + 25.161;
   1:  PR[91,3] = PR[90,3] + 75.177;
   1:L PR[91] R[100]mm/sec CNT100;
   1:  PR[91,1] = PR[90,1] + 45.035;
   1:  PR[91,2] = PR[90,2] + 25.297;
   1:  PR[91,3] = PR[90,3] + 75.195;
   1:L PR[91] R[100]mm/sec CNT100;
   1:  PR[91,1] = PR[90,1] + 44.859;
   1:  PR[91,2] = PR[90,2] + 25.339;
   1:  PR[91,3] = PR[90,3] + 75.197;
   1:L PR[91] R[100]mm/sec CNT100;
   1:  PR[91,1] = PR[90,1] + 40.843;
   1:  PR[91,2] = PR[90,2] + 26.030;
   1:  PR[91,3] = PR[90,3] + 75.198;
   1:L PR[91] R[100]mm/sec CNT100;
   1:  PR[91,1] = PR[90,1] + 37.562;
   1:  PR[91,2] = PR[90,2] + 26.283;
   1:  PR[91,3] = PR[90,3] + 75.213;
   1:L PR[91] R[100]mm/sec CNT100;
   1:  PR[91,1] = PR[90,1] + 36.092;
   1:  PR[91,2] = PR[90,2] + 26.308;
   1:  PR[91,3] = PR[90,3] + 75.225;
   1:L PR[91] R[100]mm/sec CNT100;
   1:  PR[91,1] = PR[90,1] + 30.917;
   1:  PR[91,2] = PR[90,2] + 25.890;
   1:  PR[91,3] = PR[90,3] + 75.231;
   1:L PR[91] R[100]mm/sec CNT100;
   1:  PR[91,1] = PR[90,1] + 30.362;
   1:  PR[91,2] = PR[90,2] + 25.763;
   1:  PR[91,3] = PR[90,3] + 75.251;
   1:L PR[91] R[100]mm/sec CNT100;
   1:  PR[91,1] = PR[90,1] + 25.698;
   1:  PR[91,2] = PR[90,2] + 24.546;
   1:  PR[91,3] = PR[90,3] + 75.253;
   1:L PR[91] R[100]mm/sec CNT100;
   1:  PR[91,1] = PR[90,1] + 23.070;
   1:  PR[91,2] = PR[90,2] + 24.943;
   1:  PR[91,3] = PR[90,3] + 75.271;
   1:L PR[91] R[100]mm/sec CNT100;
   1:  PR[91,1] = PR[90,1] + 18.784;
   1:  PR[91,2] = PR[90,2] + 25.081;
   1:  PR[91,3] = PR[90,3] + 75.281;
   1:L PR[91] R[100]mm/sec CNT100;
   1:  PR[91,1] = PR[90,1] + 16.908;
   1:  PR[91,2] = PR[90,2] + 25.005;
   1:  PR[91,3] = PR[90,3] + 75.298;
   1:L PR[91] R[100]mm/sec CNT100;
   1:  PR[91,1] = PR[90,1] + 12.259;
   1:  PR[91,2] = PR[90,2] + 24.002;
   1:  PR[91,3] = PR[90,3] + 75.305;
   1:L PR[91] R[100]mm/sec CNT100;
   1:  PR[91,1] = PR[90,1] + 10.802;
   1:  PR[91,2] = PR[90,2] + 23.605;
   1:  PR[91,3] = PR[90,3] + 75.323;
   1:L PR[91] R[100]mm/sec CNT100;
   1:  PR[91,1] = PR[90,1] + 8.886;
   1:  PR[91,2] = PR[90,2] + 22.726;
   1:  PR[91,3] = PR[90,3] + 75.328;
   1:L PR[91] R[100]mm/sec CNT100;
   1:  PR[91,1] = PR[90,1] + 5.324;
   1:  PR[91,2] = PR[90,2] + 23.643;
   1:  PR[91,3] = PR[90,3] + 75.336;
   1:L PR[91] R[100]mm/sec CNT100;
   1:  PR[91,1] = PR[90,1] + 5.104;
   1:  PR[91,2] = PR[90,2] + 23.687;
   1:  PR[91,3] = PR[90,3] + 75.350;
   1:L PR[91] R[100]mm/sec CNT100;
   1:  PR[91,1] = PR[90,1] + 3.617;
   1:  PR[91,2] = PR[90,2] + 23.863;
   1:  PR[91,3] = PR[90,3] + 75.351;
   1:L PR[91] R[100]mm/sec CNT100;
   1:  PR[91,1] = PR[90,1] + -2.282;
   1:  PR[91,2] = PR[90,2] + 24.280;
   1:  PR[91,3] = PR[90,3] + 75.357;
   1:L PR[91] R[100]mm/sec CNT100;
   1:  PR[91,1] = PR[90,1] + -8.620;
   1:  PR[91,2] = PR[90,2] + 23.673;
   1:  PR[91,3] = PR[90,3] + 75.379;
   1:L PR[91] R[100]mm/sec CNT100;
   1:  PR[91,1] = PR[90,1] + -11.209;
   1:  PR[91,2] = PR[90,2] + 23.066;
   1:  PR[91,3] = PR[90,3] + 75.403;
   1:L PR[91] R[100]mm/sec CNT100;
   1:  PR[91,1] = PR[90,1] + -13.126;
   1:  PR[91,2] = PR[90,2] + 23.328;
   1:  PR[91,3] = PR[90,3] + 75.413;
   1:L PR[91] R[100]mm/sec CNT100;
   1:  PR[91,1] = PR[90,1] + -16.975;
   1:  PR[91,2] = PR[90,2] + 23.749;
   1:  PR[91,3] = PR[90,3] + 75.421;
   1:L PR[91] R[100]mm/sec CNT100;
   1:  PR[91,1] = PR[90,1] + -19.485;
   1:  PR[91,2] = PR[90,2] + 23.979;
   1:  PR[91,3] = PR[90,3] + 75.436;
   1:L PR[91] R[100]mm/sec CNT100;
   1:  PR[91,1] = PR[90,1] + -29.474;
   1:  PR[91,2] = PR[90,2] + 24.347;
   1:  PR[91,3] = PR[90,3] + 75.445;
   1:L PR[91] R[100]mm/sec CNT100;
   1:  PR[91,1] = PR[90,1] + -34.147;
   1:  PR[91,2] = PR[90,2] + 24.216;
   1:  PR[91,3] = PR[90,3] + 75.483;
   1:L PR[91] R[100]mm/sec CNT100;
   1:  PR[91,1] = PR[90,1] + -38.113;
   1:  PR[91,2] = PR[90,2] + 23.878;
   1:  PR[91,3] = PR[90,3] + 75.501;
   1:L PR[91] R[100]mm/sec CNT100;
   1:  PR[91,1] = PR[90,1] + -41.302;
   1:  PR[91,2] = PR[90,2] + 23.667;
   1:  PR[91,3] = PR[90,3] + 75.516;
   1:L PR[91] R[100]mm/sec CNT100;
   1:  PR[91,1] = PR[90,1] + -47.543;
   1:  PR[91,2] = PR[90,2] + 22.599;
   1:  PR[91,3] = PR[90,3] + 75.528;
   1:L PR[91] R[100]mm/sec CNT100;
   1:  PR[91,1] = PR[90,1] + -48.481;
   1:  PR[91,2] = PR[90,2] + 22.419;
   1:  PR[91,3] = PR[90,3] + 75.552;
   1:L PR[91] R[100]mm/sec CNT100;
   1:  PR[91,1] = PR[90,1] + -53.662;
   1:  PR[91,2] = PR[90,2] + 20.734;
   1:  PR[91,3] = PR[90,3] + 75.556;
   1:L PR[91] R[100]mm/sec CNT100;
   1:  PR[91,1] = PR[90,1] + -56.367;
   1:  PR[91,2] = PR[90,2] + 19.749;
